modbus_var : ARRAY[0..100] OF INT;
modbus_var_1000 : ARRAY[0..123] OF WORD;
modbus_var_1001 : ARRAY[124..247] OF WORD;
modbus_var_1002 : ARRAY[248..371] OF WORD;
{attribute 'ac_datalog_hysteresis' := '0.2'}
{attribute 'ac_datalog' := 'DatalogChannel_4'}
Temp_chilled_medium_out : REAL;
{attribute 'ac_datalog_hysteresis' := '0.2'}
{attribute 'ac_datalog' := 'DatalogChannel_4'}
Temp_chilled_medium_in : REAL;
{attribute 'ac_datalog_hysteresis' := '0.2'}
{attribute 'ac_datalog' := 'DatalogChannel_4'}
Temp_water_inlet_cond : REAL;
{attribute 'ac_datalog_hysteresis' := '0.2'}
{attribute 'ac_datalog' := 'DatalogChannel_4'}
Press_suction_compr : REAL;
{attribute 'ac_datalog_hysteresis' := '0.5'}
{attribute 'ac_datalog' := 'DatalogChannel_4'}
Press_discharge_compr : REAL;
{attribute 'ac_datalog_hysteresis' := '0.5'}
{attribute 'ac_datalog' := 'DatalogChannel_4'}
Press_oil_receiver : REAL;
{attribute 'ac_datalog_hysteresis' := '0.5'}
{attribute 'ac_datalog' := 'DatalogChannel_4'}
Press_oil_compr : REAL;
{attribute 'ac_datalog_hysteresis' := '0.4'}
{attribute 'ac_datalog' := 'DatalogChannel_4'}
Temp_discharge : REAL;
{attribute 'ac_datalog_hysteresis' := '0.5'}
{attribute 'ac_datalog' := 'DatalogChannel_4'}
Oil_temp_receiver : REAL;
{attribute 'ac_datalog_hysteresis' := '0.5'}
{attribute 'ac_datalog' := 'DatalogChannel_4'}
Max_motor_temp : REAL;
{attribute 'ac_datalog_hysteresis' := '0.2'}
{attribute 'ac_datalog' := 'DatalogChannel_4'}
Temp_motor_bearing_DE : REAL;
{attribute 'ac_datalog_hysteresis' := '0.2'}
{attribute 'ac_datalog' := 'DatalogChannel_4'}
Temp_motor_bearing_NDE : REAL;
{attribute 'ac_datalog_hysteresis' := '4'}
{attribute 'ac_datalog' := 'DatalogChannel_4'}
Motor_current : REAL;
{attribute 'ac_datalog_hysteresis' := '50'}
{attribute 'ac_datalog' := 'DatalogChannel_4'}
Running_hours_comp_unscaled : WORD;
{attribute 'ac_datalog_hysteresis' := '50'}
{attribute 'ac_datalog' := 'DatalogChannel_4'}
Running_hours_oil_pump_unscaled : WORD;
{attribute 'ac_datalog' := 'DatalogChannel_4'}
Anti_recycle_time : REAL;
{attribute 'ac_datalog_hysteresis' := '2'}
{attribute 'ac_datalog' := 'DatalogChannel_4'}
Feedback_compressor : REAL;
{attribute 'ac_datalog_hysteresis' := '0.2'}
{attribute 'ac_datalog' := 'DatalogChannel_4'}
Oil_diff_pressure : REAL;
{attribute 'ac_datalog_hysteresis' := '0.3'}
{attribute 'ac_datalog' := 'DatalogChannel_4'}
Suction_saturated_temp : REAL;
{attribute 'ac_datalog_hysteresis' := '0.2'}
{attribute 'ac_datalog' := 'DatalogChannel_4'}
Discharge_saturated_temp : REAL;
{attribute 'ac_datalog_hysteresis' := '0.2'}
{attribute 'ac_datalog' := 'DatalogChannel_4'}
Temp_water_outlet_cond : REAL;
{attribute 'ac_datalog_hysteresis' := '0.2'}
{attribute 'ac_datalog' := 'DatalogChannel_4'}
Temp_motor_wind_R : REAL;
{attribute 'ac_datalog_hysteresis' := '0.2'}
{attribute 'ac_datalog' := 'DatalogChannel_4'}
Temp_motor_wind_S : REAL;
{attribute 'ac_datalog_hysteresis' := '0.2'}
{attribute 'ac_datalog' := 'DatalogChannel_4'}
Temp_motor_wind_T : REAL;
{attribute 'ac_datalog_hysteresis' := '0.2'}
{attribute 'ac_datalog' := 'DatalogChannel_4'}
Temp_motor_air : REAL;
{attribute 'ac_datalog_hysteresis' := '0.04'}
{attribute 'ac_datalog' := 'DatalogChannel_4'}
dP_CW : REAL;
{attribute 'ac_datalog_hysteresis' := '0.04'}
{attribute 'ac_datalog' := 'DatalogChannel_4'}
dP_SW : REAL;
{attribute 'ac_datalog_hysteresis' := '4'}
{attribute 'ac_datalog' := 'DatalogChannel_4'}
Chiller_capacity : REAL;
{attribute 'ac_datalog_hysteresis' := '2'}
{attribute 'ac_datalog' := 'DatalogChannel_4'}
Temp_oil_inlet_compr : REAL;
Spare : REAL;
{attribute 'ac_datalog_hysteresis' := '2'}
{attribute 'ac_datalog' := 'DatalogChannel_4'}
SP_CW_controller : REAL;
{attribute 'ac_datalog_hysteresis' := '2'}
{attribute 'ac_datalog' := 'DatalogChannel_4'}
Setpoint_oil_pump : REAL;
{attribute 'ac_datalog_hysteresis' := '0.02'}
{attribute 'ac_datalog' := 'DatalogChannel_4'}
Thrust_bearing_position : REAL;
{attribute 'ac_datalog_hysteresis' := '50'}
{attribute 'ac_datalog' := 'DatalogChannel_4'}
Oil_pump_running_hours : REAL;
{attribute 'ac_datalog_hysteresis' := '5'}
{attribute 'ac_datalog' := 'DatalogChannel_4'}
Liquid_level_condenser : REAL;
{attribute 'ac_datalog_hysteresis' := '0.05'}
{attribute 'ac_datalog' := 'DatalogChannel_4'}
Oil_Filter_Drop : REAL; 
{attribute 'ac_datalog_hysteresis' := '2'}
{attribute 'ac_datalog' := 'DatalogChannel_4'}
Proximitor_thrust_pos : REAL;
{attribute 'ac_datalog_hysteresis' := '0.4'}
{attribute 'ac_datalog' := 'DatalogChannel_4'}
Press_chilled_medium_in : REAL;
{attribute 'ac_datalog_hysteresis' := '0.2'}
{attribute 'ac_datalog' := 'DatalogChannel_4'}
Press_water_cond_out : REAL;
{attribute 'ac_datalog_hysteresis' := '0.02'}
{attribute 'ac_datalog' := 'DatalogChannel_4'}
Feedback_sea_water_valve : REAL;
{attribute 'ac_datalog_hysteresis' := '1'}
{attribute 'ac_datalog' := 'DatalogChannel_4'}
Oil_pressure_before_filter : REAL;
{attribute 'ac_datalog_hysteresis' := '0.2'}
{attribute 'ac_datalog' := 'DatalogChannel_4'}
Trafo_winding_temp : REAL;
{attribute 'ac_datalog_hysteresis' := '1'}
{attribute 'ac_datalog' := 'DatalogChannel_4'}
Feedback_VGD : REAL;
{attribute 'ac_datalog_hysteresis' := '4'}
{attribute 'ac_datalog' := 'DatalogChannel_4'}
Feedback_liquid_valve : REAL;
{attribute 'ac_datalog_hysteresis' := '3'}
{attribute 'ac_datalog' := 'DatalogChannel_4'}
Feedback_HGV : REAL;
{attribute 'ac_datalog_hysteresis' := '2'}
{attribute 'ac_datalog' := 'DatalogChannel_4'}
Discharge_superheat : REAL;
{attribute 'ac_datalog_hysteresis' := '0.6'}
{attribute 'ac_datalog' := 'DatalogChannel_4'}
Frequency_oil_pump : REAL;
{attribute 'ac_datalog_hysteresis' := '3'}
{attribute 'ac_datalog' := 'DatalogChannel_4'}
Hot_gas_valve_output : REAL;
{attribute 'ac_datalog_hysteresis' := '2'}
{attribute 'ac_datalog' := 'DatalogChannel_4'}
Control_signal_unit_d : REAL;
{attribute 'ac_datalog_hysteresis' := '2'}
{attribute 'ac_datalog' := 'DatalogChannel_4'}
Stall_detector : REAL;
{attribute 'ac_datalog_hysteresis' := '0.2'}
{attribute 'ac_datalog' := 'DatalogChannel_4'}
SP_MC_controller : REAL;
{attribute 'ac_datalog_hysteresis' := '2'}
{attribute 'ac_datalog' := 'DatalogChannel_4'}
Prerotary_output : REAL;
{attribute 'ac_datalog_hysteresis' := '2'}
{attribute 'ac_datalog' := 'DatalogChannel_4'}
VGD_output : REAL;
{attribute 'ac_datalog_hysteresis' := '2'}
{attribute 'ac_datalog' := 'DatalogChannel_4'}
SP_PID_compressor : REAL;
{attribute 'ac_datalog_hysteresis' := '2'}
{attribute 'ac_datalog' := 'DatalogChannel_4'}
Output_PID_suction : REAL;
{attribute 'ac_datalog_hysteresis' := '2'}
{attribute 'ac_datalog' := 'DatalogChannel_4'}
Output_PID_discharge : REAL;
{attribute 'ac_datalog_hysteresis' := '2'}
{attribute 'ac_datalog' := 'DatalogChannel_4'}
Output_PID_motor : REAL;
{attribute 'ac_datalog_hysteresis' := '2'}
{attribute 'ac_datalog' := 'DatalogChannel_4'}
Output_PID_superheat : REAL;
{attribute 'ac_datalog_hysteresis' := '2'}
{attribute 'ac_datalog' := 'DatalogChannel_4'}
SP_control : REAL;
{attribute 'ac_datalog_hysteresis' := '2'}
{attribute 'ac_datalog' := 'DatalogChannel_4'}
Unit_control_signal : REAL;
{attribute 'ac_datalog_hysteresis' := '2'}
{attribute 'ac_datalog' := 'DatalogChannel_4'}
Feedback_PRV : REAL;
{attribute 'ac_datalog_hysteresis' := '0.3'}
{attribute 'ac_datalog' := 'DatalogChannel_4'}
Theta_out : REAL;
{attribute 'ac_datalog_hysteresis' := '50'}
{attribute 'ac_datalog' := 'DatalogChannel_4'}
Alarm_limit_stall_count_unscaled : WORD;
{attribute 'ac_datalog_hysteresis' := '50'}
{attribute 'ac_datalog' := 'DatalogChannel_4'}
Alarm_limit_stall_count : REAL;
{attribute 'ac_datalog_hysteresis' := '2'}
{attribute 'ac_datalog' := 'DatalogChannel_4'}
Stall_ramp : REAL;
Min_allowed_PRVposition : REAL;
Number_of_starts : REAL;
SP_freq_oil_pump_VFD : REAL;
SP_oil_pressure_diff : REAL;
SP_oil_pressure : REAL;
{attribute 'ac_datalog_hysteresis' := '2'}
{attribute 'ac_datalog' := 'DatalogChannel_4'}
Setpoint_conv_oil_pump : REAL;
Days_above_stall_limit : REAL;
Hrs_above_stall_limit : REAL;
Min_above_stall_limit : REAL;
Sec_above_stall_limit : REAL;
{attribute 'ac_datalog_hysteresis' := '2'}
{attribute 'ac_datalog' := 'DatalogChannel_4'}
SP_cond_press : REAL;
{attribute 'ac_datalog_hysteresis' := '2'}
{attribute 'ac_datalog' := 'DatalogChannel_4'}
SP_PID_Level : REAL;
{attribute 'ac_datalog_hysteresis' := '2'}
{attribute 'ac_datalog' := 'DatalogChannel_4'}
Control_signal_SW_valve : REAL;
{attribute 'ac_datalog_hysteresis' := '4'}
{attribute 'ac_datalog' := 'DatalogChannel_4'}
Liquid_valve_output : REAL;
{attribute 'ac_datalog_hysteresis' := '0.2'}
{attribute 'ac_datalog' := 'DatalogChannel_4'}
SP_PID_seawater : REAL;
{attribute 'ac_datalog_hysteresis' := '4'}
{attribute 'ac_datalog' := 'DatalogChannel_4'}
Chiller_capacity_t1 : REAL;
{attribute 'ac_datalog_hysteresis' := '2'}
{attribute 'ac_datalog' := 'DatalogChannel_4'}
SW_pump_speed_order : REAL;
{attribute 'ac_datalog_hysteresis' := '0.4'}
{attribute 'ac_datalog' := 'DatalogChannel_4'}
Press_chilled_medium_out : REAL;
{attribute 'ac_datalog_hysteresis' := '50'}
{attribute 'ac_datalog' := 'DatalogChannel_4'}
Running_hours_compressormotor : REAL;
{attribute 'ac_datalog_hysteresis' := '0.2'}
{attribute 'ac_datalog' := 'DatalogChannel_4'}
Press_water_cond_inlet : REAL;
{attribute 'ac_datalog_hysteresis' := '2'}
{attribute 'ac_datalog' := 'DatalogChannel_4'}
Speed_feedback_VFD : REAL;
{attribute 'ac_datalog_hysteresis' := '2'}
{attribute 'ac_datalog' := 'DatalogChannel_4'}
Order_VFD_perc : REAL;
{attribute 'ac_datalog_hysteresis' := '2'}
{attribute 'ac_datalog' := 'DatalogChannel_4'}
Order_VFD_Hz : REAL;
{attribute 'ac_datalog_hysteresis' := '2'}
{attribute 'ac_datalog' := 'DatalogChannel_4'}
Temp_trafo_wind_U : REAL;
{attribute 'ac_datalog_hysteresis' := '0.2'}
{attribute 'ac_datalog' := 'DatalogChannel_4'}
Temp_trafo_wind_V : REAL;
{attribute 'ac_datalog_hysteresis' := '0.2'}
{attribute 'ac_datalog' := 'DatalogChannel_4'}
Temp_trafo_wind_W : REAL;
{attribute 'ac_datalog_hysteresis' := '2'}
{attribute 'ac_datalog' := 'DatalogChannel_4'}
Opt_speed_VFD_perc : REAL;
{attribute 'ac_datalog_hysteresis' := '2'}
{attribute 'ac_datalog' := 'DatalogChannel_4'}
Opt_speed_VFD_Hz : REAL;
Surge_counter_VFD : REAL;
Spare_4 : REAL;
Spare_3 : REAL;
Spare_2 : REAL;
Spare_0 : REAL;
Vibration_compressor_DE: REAL;
Vibration_compressor_NDE: REAL;
Feedback_seawater_valve_overboard : REAL;
Feedback_seawater_valve_bypass : REAL;
CW_flow_m3: REAL;
SW_flow_m3: REAL;
Max_motor_wind_temp: REAL;
Order_SWW_overboard: REAL;
Order_SWW_bypass: REAL;
{attribute 'ac_datalog_hysteresis' := '0.4'}
{attribute 'ac_datalog' := 'DatalogChannel'}
COP_chiller_mech : REAL ;
{attribute 'ac_datalog_hysteresis' := '50'}
{attribute 'ac_datalog' := 'DatalogChannel'}
P2_mot_1_kW : REAL ;
{attribute 'ac_datalog_hysteresis' := '50'}
{attribute 'ac_datalog' := 'DatalogChannel'}
P1_motor_kW : REAL ;
{attribute 'ac_datalog_hysteresis' := '0.4'}
{attribute 'ac_datalog' := 'DatalogChannel'}
COP_chiller_ele : REAL ;
{attribute 'ac_datalog_hysteresis' := '0.2'}
{attribute 'ac_datalog' := 'DatalogChannel'}
PI_chiller : REAL ;
;{attribute 'ac_datalog_hysteresis' := '40'}
{attribute 'ac_datalog' := 'DatalogChannel'}
Wasted_energy_kW : REAL ;
{attribute 'ac_datalog_hysteresis' := '200'}
{attribute 'ac_datalog' := 'DatalogChannel'}
Chiller_capacity_kW : REAL;
Thrust_bearing_ref_min : REAL ;
Thrust_bearing_ref_max : REAL ;
Thrust_bearing_ref : REAL ;
Q2_chillerMWh : REAL ;
Chiller_P1_MWh : REAL ;
Cal_date_MMYY : REAL ;
Chiller_P2_MWh : REAL ;
Liquid_line_temp : REAL ;
VFD_motor_current : REAL ;
Feedback_liquid_valve_raw : REAL ;
Feedback_VGD_raw : REAL ;
Feedback_PRV_raw : REAL ;
Feedback_HGV_raw : REAL ;
Feedback_seawater_valve_overboard_raw : REAL ;
Feedback_seawater_valve_bypass_raw : REAL ;
SP_cond_press_limit : REAL ;
SP_evap_press_limit : REAL ;
SP_discharge_superheat_limit : REAL ;
SP_t1 : REAL ;
VFD_min_allowed_frequence : REAL ;
VFD_min_allowed_speed : REAL ;

Trip_BITs_0_to_15 : WORD;
Trip_BITs_16_to_31: WORD;
Trip_BITs_32_to_47: WORD;
Trip_BITs_48_to_63: WORD;
Trip_BITs_64_to_79: WORD;
Trip_BITs_80_to_95: WORD;
Trip_BITs_96_to_121: WORD;
Trip_BITs_122_to_137: WORD;
Trip_BITs_138_to_153: WORD;
Trip_BITs_154_to_169: WORD;
Trip_BITs_170_to_185: WORD;
Trip_BITs_186_to_201: WORD;


Alarm_BITs_0_to_15: WORD;
Alarm_BITs_16_to_31: WORD;
Alarm_BITs_32_to_47: WORD;
Alarm_BITs_48_to_63: WORD;
Alarm_BITs_64_to_79: WORD;
Alarm_BITs_80_to_95: WORD;
Alarm_BITs_96_to_111: WORD;

Status_BITs_0_to_15 : WORD;
Status_BITs_16_to_31 : WORD;
Status_BITs_32_to_47: WORD;
Status_BITs_48_to_63: WORD;
Status_BITs_64_to_79: WORD;
Status_BITs_80_to_95: WORD;
Status_BITs_96_to_111: WORD;
Status_BITs_112_to_127: WORD;




DI_Status_BITs_0_to_15 : WORD;
DI_Status_BITs_16_to_31: WORD;

DO_Status_BITs_16_to_31: WORD;
DO_Status_BITs_32_to_47: WORD;

T_Overload_compressor_motor : BOOL;
T_Compressor_running_failure : BOOL;
T_Low_chilled_medium_outlet : BOOL;
T_Low_sea_water_flow : BOOL;
T_Oil_level_motor_bearing : BOOL;

T_Low_oil_flow : BOOL;
T_Overload_oil_pump_motor : BOOL;
T_Oil_pump_running_failure : BOOL;
T_Low_oil_flow_trip : BOOL;
T_High_temp_oil_receiver : BOOL;
T_Low_temp_oil_receiver : BOOL;
T_Low_suction_pressure : BOOL;
T_High_suction_pressure : BOOL;
T_High_discharge_pressure : BOOL;
T_Low_discharge_pressure : BOOL;
T_High_discharge_temp : BOOL;
T_Low_oil_diff_pressure : BOOL;
T_High_diff_oil_pressure : BOOL;
T_Starting_to_long : BOOL;
T_Surge_detection : BOOL;
T_Comp_thrust_bearing_position : BOOL;
Spare_trip_1 : BOOL;
T_Chilled_pump_run_failure : BOOL;
T_Sea_water_pump_run_failure : BOOL;
T_Low_chilled_medium_flow : BOOL;
T_High_chilled_medium_flow : BOOL;
T_Low_condenser_flow : BOOL;
T_High_condenser_flow : BOOL;
T_Emergency_stop : BOOL;
T_High_comp_mot_DE_bear_temp : BOOL;
T_High_comp_mot_NDE_bear_temp : BOOL;
T_High_motor_air_temp : BOOL;
T_Comp_motor_leak_detection : BOOL;
T_High_comp_mot_DE_bear_vib : BOOL;
T_High_comp_mot_NDE_bear_Vib : BOOL;
T_High_comp_motor_wind_temp : BOOL;
Spare_trip_2 : BOOL;
T_Rotating_stall_trip : BOOL;
T_Analog_inputs : BOOL;
T_Feedback_CW_valve : BOOL;
T_Low_oil_diff_press_prelub : BOOL;
T_Low_oil_diff_press_standstil : BOOL;

T_Spare_3 : BOOL;
T_Spare_4 : BOOL;
T_Spare_5 : BOOL;
T_Spare_6 : BOOL;
T_Spare_7 : BOOL;
T_Spare_8 : BOOL;
T_High_temp_oil_inlet_comp : BOOL;
T_Comp_motor_power_loss : BOOL;
Spare_trip_3 : BOOL;
T_Cathodic_protect_sys_alarm : BOOL;
T_High_oil_filter_diff_press : BOOL;
T_Flow_switch_FT01 : BOOL;
T_Starter_failure_trip : BOOL;
T_Incorrect_feedback_starter_trip : BOOL;

A_VGD_fault : BOOL;
A_High_condenser_flow : BOOL;
A_Rotating_stall : BOOL;
A_High_temp_oil_inlet_comp : BOOL;
SpareAlarm_1 : BOOL;
A_High_motor_air_temp : BOOL;
A_High_control_panel_temp : BOOL;
A_Low_oil_diff_pressure : BOOL;
Spare_alarm_2 : BOOL;
A_High_comp_motor_winding_temp : BOOL;
A_High_comp_mo_DE_bear_temp : BOOL;
A_High_comp_mo_NDE_bear_temp : BOOL;
A_High_comp_mo_DE_bear_vib : BOOL;
A_High_comp_mo_NDE_bear_vib : BOOL;
A_Low_chilled_medium_flow : BOOL;
A_High_chilled_medium_flow : BOOL;
A_Low_sea_water_flow : BOOL;
A_Seawater_pump_not_running : BOOL;
A_Spare : BOOL;
A_Spare_1 : BOOL;
A_Spare_2 : BOOL;
A_Spare_3 : BOOL;
A_Spare_4 : BOOL;
A_Spare_5 : BOOL;
A_Spare_6 : BOOL;
A_Spare_7 : BOOL;
A_Spare_8 : BOOL;
A_Spare_9 : BOOL;
A_Spare_10 : BOOL;
A_Spare_11 : BOOL;
A_High_oil_filter_diff_press : BOOL;
A_Spare_12 : BOOL;
A_Spare_13 : BOOL;
A_Spare_14 : BOOL;
A_Spare_15 : BOOL;
A_Spare_16 : BOOL;
A_Spare_17 : BOOL;
Anti_recycle_status : BOOL;
Low_oil_temperature : BOOL;
Low_oil_temp_auto : BOOL;
Oil_heater : BOOL;
Sea_water_pump : BOOL;
Comp_oil_pump : BOOL;
Bearing_oil_pump : BOOL;
Solenoid_oil_return : BOOL;
Unit_running : BOOL;
Unit_remote : BOOL;
Unit_auto : BOOL;
Unit_manual : BOOL;
Unit_trip : BOOL;
Unit_alarm : BOOL;
Unit_start_switch : BOOL;
Unit_available : BOOL;
Unit_fault : BOOL;
S_Spare_1 : BOOL;
S_Spare_2 : BOOL;
S_Spare_3 : BOOL;
S_Spare_4 : BOOL;
S_Spare_5 : BOOL;
S_Spare_6 : BOOL;
S_Spare_7 : BOOL;
S_Spare_8 : BOOL;
Solenoid_liquid_inj: BOOL;
CW_Flow_ind : BOOL;
Open_chilled_water_valve : BOOL;
Feedback_chilled_water_valve : BOOL;
Open_order_swv_overboard : BOOL;
Close_order_swv_overboard : BOOL;
Open_order_swv_bypass : BOOL;
Close_order_swv_bypass : BOOL;
VFD_man_auto : BOOL ;
VFD_freq_jump_on : BOOL ;
VFD_ramp_100_perc : BOOL ;
VFD_locked_100_perc : BOOL;
VFD_ramp_d_PRVcontrol : BOOL;
PRV_control : BOOL;
VFD_control : BOOL;
VFD_fixed_speed : BOOL;
Spare_151: BOOL;
T_Transformer_winding_temp : BOOL;
A_Transformer_winding_temp : BOOL;
T_trafo_opening_main_breaker : BOOL;
T_VFD : BOOL;
VFD_ready : BOOL;
T_VFD_emergency_stop : BOOL;
T_Low_5VDC_supply : BOOL;
T_High_5VDC_supply : BOOL;
T_Spare_9 : BOOL;
T_Spare_10 : BOOL;
T_Spare_11 : BOOL;
T_Spare_12 : BOOL;
T_Spare_13 : BOOL;
T_Low_liquid_level : BOOL;
T_SW_pump_off_to_long : BOOL;
T_Softstarter_failure : BOOL;
T_Motorstarter_failure : BOOL ;
T_CW_valveopen_failure : BOOL ;
T_SW_valveopen_failure : BOOL ;
T_High_disch_superheat :BOOL ;
T_Low_disch_superheat :BOOL ;
T_High_CW_outlet_temp : BOOL;
T_Low_CW_outlet_temp : BOOL;
T_Low_CW_inlet_temp : BOOL;
T_High_CW_inlet_temp : BOOL;
T_High_SW_outlet_temp : BOOL;
T_Low_SW_outlet_temp : BOOL;
T_Low_SW_inlet_temp : BOOL;
T_High_SW_inlet_temp : BOOL;
T_High_motor_wind_temp_R : BOOL;
T_High_motor_wind_temp_S : BOOL;
T_High_motor_wind_temp_T : BOOL;
T_High_press_ratio : BOOL;
T_Low_press_ratio : BOOL;
T_Low_CW_dP : BOOL;
T_High_CW_dP : BOOL;
T_Low_SW_dP : BOOL;
T_High_SW_dP : BOOL;
T_Long_time_PRV : BOOL;
T_Comp_thrust_neg_move : BOOL;
T_Comp_thrust_pos_move : BOOL;
T_VGD_fault : BOOL;
T_Low_oilpress_prelube : BOOL;
T_Low_temp_oil_inlet_comp : BOOL;
T_Low_oilpress_standby : BOOL;
T_Rotating_stall : BOOL;

T_Sensor_failure_AI_128: BOOL;
T_Sensor_failure_AI_130: BOOL;
T_Sensor_failure_AI_134: BOOL;
T_Sensor_failure_AI_256: BOOL;
T_Sensor_failure_AI_258: BOOL;
T_Sensor_failure_AI_260: BOOL;
T_Sensor_failure_AI_262: BOOL;
T_Sensor_failure_AI_264: BOOL;
T_Sensor_failure_AI_266: BOOL;
T_Sensor_failure_AI_268: BOOL;
T_Sensor_failure_AI_270: BOOL;
T_Sensor_failure_AI_272: BOOL;
T_Sensor_failure_AI_274: BOOL;
T_Sensor_failure_AI_276: BOOL;
T_Sensor_failure_AI_278: BOOL;
T_Sensor_failure_AI_280: BOOL;
T_Sensor_failure_AI_282: BOOL;
T_Sensor_failure_AI_284: BOOL;
T_Sensor_failure_AI_286: BOOL;
T_Sensor_failure_AI_288: BOOL;
T_Sensor_failure_AI_290: BOOL;
T_Sensor_failure_AI_292: BOOL;
T_Sensor_failure_AI_294: BOOL;
T_Sensor_failure_AI_296: BOOL;
T_Sensor_failure_AI_298: BOOL;
T_Sensor_failure_AI_330: BOOL;
T_Sensor_failure_AI_320: BOOL;
T_Sensor_failure_AI_322: BOOL;
T_Sensor_failure_AI_324: BOOL;
T_Sensor_failure_AI_326: BOOL;
T_Sensor_failure_AI_328: BOOL;
T_Sensor_failure_AI_332: BOOL;
T_Sensor_failure_AI_334: BOOL;
T_Sensor_failure_AI_300: BOOL;
T_Sensor_failure_AI_302: BOOL;
T_Sensor_failure_AI_304: BOOL;
T_Sensor_failure_AI_306: BOOL;
T_Sensor_failure_AI_308: BOOL;
T_Sensor_failure_AI_310: BOOL;
T_Sensor_failure_AI_312: BOOL;
T_Sensor_failure_AI_314: BOOL;
T_Sensor_failure_AI_316: BOOL;
T_Sensor_failure_AI_318: BOOL;
T_Sensor_failure_AI_352: BOOL;
T_Sensor_failure_AI_354: BOOL;
T_Sensor_failure_AI_360: BOOL;
T_Sensor_failure_AI_362: BOOL;
T_Sensor_failure_AI_364: BOOL;
T_Sensor_failure_AI_368: BOOL;
T_Sensor_failure_AI_370: BOOL;
T_Sensor_failure_AI_372: BOOL;
T_Sensor_failure_AI_374: BOOL;
T_Sensor_failure_AI_376: BOOL;
T_Sensor_failure_AI_378: BOOL;
T_Sensor_failure_AI_380: BOOL;
T_Sensor_failure_AI_382: BOOL;
T_Sensor_failure_AI_336: BOOL;
T_Sensor_failure_AI_338: BOOL;
T_Sensor_failure_AI_340: BOOL;
T_Sensor_failure_AI_342: BOOL;
T_Sensor_failure_AI_344: BOOL;
T_Sensor_failure_AI_346: BOOL;
T_Sensor_failure_AI_348: BOOL;
T_Sensor_failure_AI_350: BOOL;
T_Sensor_failure_AI_752: BOOL;
T_Sensor_failure_AI_754: BOOL;
T_Sensor_failure_AI_756: BOOL;
T_Sensor_failure_AI_760: BOOL;
T_Sensor_failure_AI_772: BOOL;
T_Sensor_failure_AI_774: BOOL;
T_Sensor_failure_AI_776: BOOL;
T_Sensor_failure_AI_778: BOOL;
T_Sensor_failure_AI_780: BOOL;

A_high_disch_press : BOOL ;
A_low_disch_press : BOOL ;
A_Low_suction_pressure : BOOL;
A_High_suction_pressure : BOOL;
A_High_discharge_temp : BOOL;
A_High_oil_temp_receiver : BOOL;
A_Low_oil_temp_receiver : BOOL;
A_Low_temp_oil_inlet_comp : BOOL;
A_High_oil_diff_pressure : BOOL;
A_Low_discharge_superheat : BOOL;
A_High_discharge_superheat : BOOL;
A_Low_CW_outlet_temp : BOOL;
A_High_CW_outlet_temp : BOOL;
A_Low_CW_inlet_temp : BOOL;
A_High_CW_inlet_temp : BOOL;
A_High_SW_outlet_temp : BOOL;
A_Low_condenser_flow : BOOL;
A_High_press_ratio : BOOL;
A_Low_press_ratio : BOOL;
A_Motor_speed_low : BOOL;
A_Low_SW_outlet_temp : BOOL;
A_Low_SW_inlet_temp : BOOL;
A_High_SW_inlet_temp : BOOL;
A_High_suction_superheat : BOOL;
A_Low_suction_superheat : BOOL;
A_High_temp_oil_separator : BOOL;
A_Low_temp_oil_separator : BOOL;
A_High_motor_wind_temp_R : BOOL;
A_High_motor_wind_temp_S : BOOL;
A_High_motor_wind_temp_T : BOOL;
A_High_CW_dP : BOOL;
A_Low_CW_dP : BOOL;
A_High_SW_dP : BOOL;
A_Low_SW_dP : BOOL;

Start_inhib_time_between_Start : BOOL;
Start_inhib_time_beetween_Stop : BOOL;
Start_inhib_PRV_not_min : BOOL;
Start_inhib_Motor_overload : BOOL;
Remote_bilge_pump_control : BOOL;
CW_pump_running : BOOL;
A_Low_liquid_level : BOOL;
A_Suction_press_limit : BOOL;
A_Discharge_press_limit : BOOL;
A_Discharge_superheat_limit : BOOL;
A_Motor_current_limit : BOOL;


DI_0_0_Emergency_stop : BOOL;
DI_0_0 : BOOL;
DI_0_1 : BOOL;
DI_0_2_Fault_reset : BOOL;
DI_0_2 : BOOL;
DI_0_3 : BOOL;
DI_0_4 : BOOL;
DI_0_5 : BOOL;
DI_0_6_Overload_protection : BOOL;
DI_0_6 : BOOL;
DI_0_7 : BOOL;
DI_1_0_Overload_oilpump : BOOL;
DI_1_0 : BOOL;
DI_1_1 : BOOL;
DI_1_2 : BOOL;
DI_1_3 : BOOL;
Power_available : BOOL;
DI_1_4 : BOOL;
DI_1_5_Starter_failure : BOOL;
DI_1_5 : BOOL;
DI_8_0_Controlpanel_temp : BOOL;
DI_8_0 : BOOL;
DI_8_1 : BOOL;
DI_8_2_VGD_limit_switch : BOOL;
DI_8_2 : BOOL;
DI_8_3_water_leak_motor  : BOOL;
DI_8_3 : BOOL;
DI_8_4_Catodic_protection : BOOL;
DI_8_4 : BOOL;
DI_8_5_Trust_bearing_probe : BOOL;
DI_8_5 : BOOL;
DI_8_6_ESD_operation : BOOL;
DI_8_6 : BOOL;
DI_8_7 : BOOL;
DI_9_0_MV_breaker_available : BOOL;
DI_9_0 : BOOL;
DI_9_1 : BOOL;
DI_9_2_Safe_return_to_port : BOOL;
DI_9_2 : BOOL;
DI_9_3 : BOOL;
DI_9_4_VFD_emergency_stop : BOOL;
DI_9_4 : BOOL;
DI_9_5 : BOOL;
DI_9_6 : BOOL;
DI_9_7 : BOOL;
DO_0_0_Start_signal_comp : BOOL;
DO_0_0 : BOOL;
DO_0_1_Start_signal_oil_pump : BOOL;
DO_0_1 : BOOL;
DO_0_2_Start_signal_SW_pump : BOOL;
DO_0_2 : BOOL;
DO_0_3_Start_signal_CW_pump : BOOL;
DO_0_3 : BOOL;
DO_0_4_Solenoid_valve_oil : BOOL;
DO_0_4 : BOOL;
DO_0_5_Solenoid_valve_liquid : BOOL;
DO_0_5 : BOOL;
DO_0_6_Oil_heater : BOOL;
DO_0_6 : BOOL;
DO_0_7_Comp_heater : BOOL;
DO_0_7 : BOOL;
DO_1_0 : BOOL;
DO_1_1 : BOOL;
DO_8_0_Liquid_valve_open : BOOL;
DO_8_0 : BOOL;
DO_8_1_Liquid_valve_close : BOOL;
DO_8_1 : BOOL;
DO_8_2_VGD_open : BOOL;
DO_8_2 : BOOL;
DO_8_3_VGD_close : BOOL;
DO_8_3 : BOOL;
DO_8_4_PRV_open : BOOL;
DO_8_4 : BOOL;
DO_8_5_PRV_close : BOOL;
DO_8_5 : BOOL;
DO_8_6_HGV_open : BOOL;
DO_8_6 : BOOL;
DO_8_7_HGV_close : BOOL;
DO_8_7 : BOOL;
DO_9_0_Open_order_swv_overboard : BOOL;
DO_9_0 : BOOL;
DO_9_1_Close_order_swv_overboard : BOOL;
DO_9_1 : BOOL;
DO_9_2_Open_order_swv_bypass : BOOL;
DO_9_2 : BOOL;
DO_9_3_Close_order_swv_bypass : BOOL;
DO_9_3 : BOOL;
DO_9_4 : BOOL;
DO_9_5 : BOOL;
DO_9_6 : BOOL;
DO_9_7 : BOOL;
Power_request : BOOL;
DO_12_0 : BOOL;
DO_12_1_Compressor_ready : BOOL;
DO_12_1 : BOOL;
DO_12_2 : BOOL;
DO_12_3 : BOOL;
DO_12_4_Control_panel_alarm : BOOL;
DO_12_4 : BOOL;
DO_12_5_Auto_reset : BOOL;
DO_12_5 : BOOL;
DO_12_6_Unit_running : BOOL;
DO_12_6 : BOOL;
DO_12_7 : BOOL;
Start_inhib_time_Oil_receiver_temp : BOOL;
PrV_in_min : BOOL;


//Graphic variables
Unit_switch_status : INT;
i : INT;
show_trendvalue : ARRAY[0..50] OF BOOL;
select_trendvalue : INT :=0 ;

END_VAR


Temp_chilled_medium_out:=scaleFunction(modbus_var_1000[10],0.1, 0);
Temp_chilled_medium_in:=scaleFunction(modbus_var_1000[11],0.1, 0);
Temp_water_inlet_cond:=scaleFunction(modbus_var_1000[12],0.1, 0);
Press_suction_compr:=scaleFunction(modbus_var_1000[13],0.01, 0);
Press_discharge_compr:=scaleFunction(modbus_var_1000[14],0.01, 0);
Press_oil_receiver:=scaleFunction(modbus_var_1000[15],0.01, 0);
Press_oil_compr:=scaleFunction(modbus_var_1000[16],0.01, 0);
Temp_discharge:=scaleFunction(modbus_var_1000[17],0.1, 0);
Oil_temp_receiver:=scaleFunction(modbus_var_1000[18],0.1, 0);
Max_motor_temp:=scaleFunction(modbus_var_1000[19],0.1, 0);
Temp_motor_bearing_DE:=scaleFunction(modbus_var_1000[20],0.1, 0);
Temp_motor_bearing_NDE:=scaleFunction(modbus_var_1000[21],0.1, 0);
Motor_current:=scaleFunction(modbus_var_1000[22],1.0, 0);
Running_hours_comp_unscaled:=modbus_var_1000[23];
//Anti_recycle_time:=scaleFunction(modbus_var_1000[24],1.0, 0);
Feedback_compressor:=scaleFunction(modbus_var_1000[25],1.0, 0);
Oil_diff_pressure:=scaleFunction(modbus_var_1000[26],0.01, 0);
Suction_saturated_temp:=scaleFunction(modbus_var_1000[27],0.1, 0);
Discharge_saturated_temp:=scaleFunction(modbus_var_1000[28],0.1, 0);
Temp_water_outlet_cond:=scaleFunction(modbus_var_1000[29],0.1, 0);
Temp_motor_wind_R:=scaleFunction(modbus_var_1000[30],0.1, 0);
Temp_motor_wind_S:=scaleFunction(modbus_var_1000[31],0.1, 0);
Temp_motor_wind_T:=scaleFunction(modbus_var_1000[32],0.1, 0);
Temp_motor_air:=scaleFunction(modbus_var_1000[33],0.1, 0);
dP_CW:=scaleFunction(modbus_var_1000[34],0.01, 0);
dP_SW:=scaleFunction(modbus_var_1000[35],0.01, 0);
CW_flow_m3:=scaleFunction(modbus_var_1000[36],1.0, 0);
Temp_oil_inlet_compr:=scaleFunction(modbus_var_1000[37],0.1, 0);
Stall_detector:=scaleFunction(modbus_var_1000[38],0.01, 0);
SP_CW_controller:=scaleFunction(modbus_var_1000[39],0.1, 0);
Feedback_sea_water_valve:=scaleFunction(modbus_var_1000[40],0.1, 0);
Oil_pressure_before_filter:=scaleFunction(modbus_var_1000[41],0.01, 0);
Feedback_VGD:=scaleFunction(modbus_var_1000[42],0.1, 0);
Chiller_capacity:=scaleFunction(modbus_var_1000[43],0.1, 0);
Setpoint_oil_pump:=scaleFunction(modbus_var_1000[44],0.01, 0);
Thrust_bearing_position:=scaleFunction(modbus_var_1000[45],0.1, 0);
Oil_pump_running_hours:=scaleFunction(modbus_var_1000[46],10, 0);
Liquid_level_condenser:=scaleFunction(modbus_var_1000[47],0.1, 0);
Oil_Filter_Drop:=scaleFunction(modbus_var_1000[48],0.01, 0);
Proximitor_thrust_pos:=scaleFunction(modbus_var_1000[49],0.1, 0);
//Spare_old_write_bits:=scaleFunction(modbus_var_1000[50],1.0, 0);
Press_chilled_medium_in:=scaleFunction(modbus_var_1000[51],0.01, 0);
Press_water_cond_out:=scaleFunction(modbus_var_1000[52],0.01, 0);
Discharge_superheat:=scaleFunction(modbus_var_1000[53],0.1, 0);
Frequency_oil_pump:=scaleFunction(modbus_var_1000[54],0.1, 0);
Feedback_liquid_valve:=scaleFunction(modbus_var_1000[55],0.1, 0);
Hot_gas_valve_output:=scaleFunction(modbus_var_1000[56],0.1, 0);
Control_signal_unit_d:=scaleFunction(modbus_var_1000[57],0.1, 0);
SP_MC_controller:=scaleFunction(modbus_var_1000[58],0.1, 0);
Prerotary_output:=scaleFunction(modbus_var_1000[59],0.1, 0);
VGD_output:=scaleFunction(modbus_var_1000[60],0.1, 0);
SP_PID_compressor:=scaleFunction(modbus_var_1000[61],0.1, 0);
Output_PID_suction:=scaleFunction(modbus_var_1000[62],0.1, 0);
Output_PID_discharge:=scaleFunction(modbus_var_1000[63],0.1, 0);
Output_PID_motor:=scaleFunction(modbus_var_1000[64],0.1, 0);
Output_PID_superheat:=scaleFunction(modbus_var_1000[65],0.1, 0);
SP_control:=scaleFunction(modbus_var_1000[66],0.1, 0);
Unit_control_signal:=scaleFunction(modbus_var_1000[67],0.1, 0);
Feedback_PRV:=scaleFunction(modbus_var_1000[68],0.1, 0);
Theta_out:=scaleFunction(modbus_var_1000[69],0.1, 0);
Alarm_limit_stall_count:=scaleFunction(modbus_var_1000[70],1.0, 0);
Stall_ramp:=scaleFunction(modbus_var_1000[71],0.1, 0);
Min_allowed_PRVposition:=scaleFunction(modbus_var_1000[72],0.1, 0);
Number_of_starts:=scaleFunction(modbus_var_1000[73],1.0, 0);
SP_oil_pressure:=scaleFunction(modbus_var_1000[74],0.01, 0);
Setpoint_conv_oil_pump:=scaleFunction(modbus_var_1000[75],0.1, 0);
Days_above_stall_limit:=scaleFunction(modbus_var_1000[76],1.0, 0);
Hrs_above_stall_limit:=scaleFunction(modbus_var_1000[77],1.0, 0);
Min_above_stall_limit:=scaleFunction(modbus_var_1000[78],1.0, 0);
Sec_above_stall_limit:=scaleFunction(modbus_var_1000[79],1.0, 0);
SP_PID_Level:=scaleFunction(modbus_var_1000[80],0.1, 0);
Control_signal_SW_valve:=scaleFunction(modbus_var_1000[81],0.1, 0);
Feedback_HGV:=scaleFunction(modbus_var_1000[82],0.1, 0);
Liquid_valve_output:=scaleFunction(modbus_var_1000[83],0.1, 0);
SP_PID_seawater:=scaleFunction(modbus_var_1000[84],0.1, 0);
Chiller_capacity_t1:=scaleFunction(modbus_var_1000[85],0.1, 0);
SW_pump_speed_order:=scaleFunction(modbus_var_1000[86],0.1, 0);
Anti_recycle_time:=scaleFunction(modbus_var_1000[87],1.0, 0);
Press_chilled_medium_out:=scaleFunction(modbus_var_1000[88],0.01, 0);
Press_water_cond_inlet:=scaleFunction(modbus_var_1000[89],0.01, 0);
Running_hours_compressormotor:=scaleFunction(modbus_var_1000[90],10, 0);

Trip_BITs_0_to_15:=modbus_var_1000[0];
Trip_BITs_16_to_31:=modbus_var_1000[1];
Trip_BITs_32_to_47:=modbus_var_1000[2];
Trip_BITs_48_to_63:=modbus_var_1000[3];
Trip_BITs_64_to_79:=modbus_var_1000[4];
// Alarm_BITs_80_to_95:=modbus_var_1000[5];
// Alarm_BITs_96_to_111:=modbus_var_1000[6];
Status_BITs_0_to_15:=modbus_var_1000[5];
Status_BITs_16_to_31:=modbus_var_1000[6];

T_Low_suction_pressure:=maskbitFunction(Trip_BITs_0_to_15,0);
T_High_discharge_pressure:=maskbitFunction(Trip_BITs_0_to_15,1);
T_High_discharge_temp:=maskbitFunction(Trip_BITs_0_to_15,2);
T_Low_oil_diff_pressure:=maskbitFunction(Trip_BITs_0_to_15,3);
T_High_diff_oil_pressure:=maskbitFunction(Trip_BITs_0_to_15,4);
T_Starting_to_long:=maskbitFunction(Trip_BITs_0_to_15,5);
T_Surge_detection:=maskbitFunction(Trip_BITs_0_to_15,6);
T_Comp_thrust_bearing_position:=maskbitFunction(Trip_BITs_0_to_15,7);
T_Overload_compressor_motor:=maskbitFunction(Trip_BITs_0_to_15,8);
T_Compressor_running_failure:=maskbitFunction(Trip_BITs_0_to_15,9);
T_Low_chilled_medium_outlet:=maskbitFunction(Trip_BITs_0_to_15,10);
T_Low_oil_flow:=maskbitFunction(Trip_BITs_0_to_15,11);
T_Overload_oil_pump_motor:=maskbitFunction(Trip_BITs_0_to_15,12);
T_Oil_pump_running_failure:=maskbitFunction(Trip_BITs_0_to_15,13);
T_Low_oil_flow_trip:=maskbitFunction(Trip_BITs_0_to_15,14);
T_High_temp_oil_receiver:=maskbitFunction(Trip_BITs_0_to_15,15);
T_High_comp_motor_wind_temp:=maskbitFunction(Trip_BITs_16_to_31,0);
T_High_comp_mot_DE_bear_temp:=maskbitFunction(Trip_BITs_16_to_31,1);
T_High_comp_mot_NDE_bear_temp:=maskbitFunction(Trip_BITs_16_to_31,2);
T_High_motor_air_temp:=maskbitFunction(Trip_BITs_16_to_31,3);
T_Comp_motor_leak_detection:=maskbitFunction(Trip_BITs_16_to_31,4);
T_High_5VDC_supply:=maskbitFunction(Trip_BITs_16_to_31,5);
T_Low_5VDC_supply:=maskbitFunction(Trip_BITs_16_to_31,6);
T_Chilled_pump_run_failure:=maskbitFunction(Trip_BITs_16_to_31,7);
T_Sea_water_pump_run_failure:=maskbitFunction(Trip_BITs_16_to_31,8);
T_Low_chilled_medium_flow:=maskbitFunction(Trip_BITs_16_to_31,9);
T_High_chilled_medium_flow:=maskbitFunction(Trip_BITs_16_to_31,10);
T_Low_sea_water_flow:=maskbitFunction(Trip_BITs_16_to_31,11);
T_High_condenser_flow:=maskbitFunction(Trip_BITs_16_to_31,12);
A_High_temp_oil_inlet_comp:=maskbitFunction(Trip_BITs_16_to_31,13);
T_Comp_motor_power_loss:=maskbitFunction(Trip_BITs_16_to_31,14);
T_Emergency_stop:=maskbitFunction(Trip_BITs_16_to_31,15);
T_Sensor_failure_AI_276:=maskbitFunction(Trip_BITs_32_to_47,0);
T_Sensor_failure_AI_278:=maskbitFunction(Trip_BITs_32_to_47,1);
T_Sensor_failure_AI_280:=maskbitFunction(Trip_BITs_32_to_47,2);
T_Sensor_failure_AI_282:=maskbitFunction(Trip_BITs_32_to_47,3);
T_Sensor_failure_AI_288:=maskbitFunction(Trip_BITs_32_to_47,4);
T_Sensor_failure_AI_292:=maskbitFunction(Trip_BITs_32_to_47,5);
T_Sensor_failure_AI_272:=maskbitFunction(Trip_BITs_32_to_47,6);
T_Sensor_failure_AI_130:=maskbitFunction(Trip_BITs_32_to_47,7);
T_Sensor_failure_AI_134:=maskbitFunction(Trip_BITs_32_to_47,8);
T_Sensor_failure_AI_128:=maskbitFunction(Trip_BITs_32_to_47,9);
T_Sensor_failure_AI_256:=maskbitFunction(Trip_BITs_32_to_47,10);
T_Sensor_failure_AI_274:=maskbitFunction(Trip_BITs_32_to_47,11);
T_Sensor_failure_AI_270:=maskbitFunction(Trip_BITs_32_to_47,12);
T_Sensor_failure_AI_268:=maskbitFunction(Trip_BITs_32_to_47,13);
T_Sensor_failure_AI_286:=maskbitFunction(Trip_BITs_32_to_47,14);
T_Sensor_failure_AI_284:=maskbitFunction(Trip_BITs_32_to_47,15);
T_Sensor_failure_AI_304:=maskbitFunction(Trip_BITs_48_to_63,0);
T_Sensor_failure_AI_308:=maskbitFunction(Trip_BITs_48_to_63,1);
T_Sensor_failure_AI_312:=maskbitFunction(Trip_BITs_48_to_63,2);
T_Sensor_failure_AI_296:=maskbitFunction(Trip_BITs_48_to_63,3);
T_Sensor_failure_AI_300:=maskbitFunction(Trip_BITs_48_to_63,4);
T_Sensor_failure_AI_316:=maskbitFunction(Trip_BITs_48_to_63,5);
T_Sensor_failure_AI_262:=maskbitFunction(Trip_BITs_48_to_63,6);
T_Sensor_failure_AI_352:=maskbitFunction(Trip_BITs_48_to_63,7);
T_Sensor_failure_AI_354:=maskbitFunction(Trip_BITs_48_to_63,8);
T_Sensor_failure_AI_360:=maskbitFunction(Trip_BITs_48_to_63,9);
T_Sensor_failure_AI_362:=maskbitFunction(Trip_BITs_48_to_63,10);
T_Sensor_failure_AI_364:=maskbitFunction(Trip_BITs_48_to_63,11);
T_Rotating_stall_trip:=maskbitFunction(Trip_BITs_48_to_63,12);
T_Analog_inputs:=maskbitFunction(Trip_BITs_48_to_63,13);
T_High_oil_filter_diff_press:=maskbitFunction(Trip_BITs_48_to_63,14);
T_Sensor_failure_AI_260:=maskbitFunction(Trip_BITs_48_to_63,15);
A_High_comp_motor_winding_temp:=maskbitFunction(Trip_BITs_64_to_79,0);
A_High_comp_mo_DE_bear_temp:=maskbitFunction(Trip_BITs_64_to_79,1);
A_High_comp_mo_NDE_bear_temp:=maskbitFunction(Trip_BITs_64_to_79,2);
A_High_motor_air_temp:=maskbitFunction(Trip_BITs_64_to_79,3);
A_Low_chilled_medium_flow:=maskbitFunction(Trip_BITs_64_to_79,4);
A_High_chilled_medium_flow:=maskbitFunction(Trip_BITs_64_to_79,5);
A_Low_sea_water_flow:=maskbitFunction(Trip_BITs_64_to_79,6);
A_High_condenser_flow:=maskbitFunction(Trip_BITs_64_to_79,7);
T_Sensor_failure_AI_258:=maskbitFunction(Trip_BITs_64_to_79,8);
T_Sensor_failure_AI_264:=maskbitFunction(Trip_BITs_64_to_79,9);
T_Sensor_failure_AI_266:=maskbitFunction(Trip_BITs_64_to_79,10);
A_Rotating_stall:=maskbitFunction(Trip_BITs_64_to_79,11);
A_Low_oil_diff_pressure:=maskbitFunction(Trip_BITs_64_to_79,12);
A_High_oil_filter_diff_press:=maskbitFunction(Trip_BITs_64_to_79,13);
A_High_control_panel_temp:=maskbitFunction(Trip_BITs_64_to_79,14);
//A_Spare:=maskbitFunction(Trip_BITs_64_to_79,15);
Unit_running:=maskbitFunction(Status_BITs_0_to_15,0);
Unit_available:=maskbitFunction(Status_BITs_0_to_15,1);
Unit_remote:=maskbitFunction(Status_BITs_0_to_15,2);
Unit_auto:=maskbitFunction(Status_BITs_0_to_15,3);
Anti_recycle_status:=maskbitFunction(Status_BITs_0_to_15,4);
//S_Spare:=maskbitFunction(Status_BITs_0_to_15,5);
//S_Spare:=maskbitFunction(Status_BITs_0_to_15,6);
//S_Spare:=maskbitFunction(Status_BITs_0_to_15,7);
//S_Spare:=maskbitFunction(Status_BITs_0_to_15,8);
Unit_trip:=maskbitFunction(Status_BITs_0_to_15,9);
Unit_alarm:=maskbitFunction(Status_BITs_0_to_15,10);
Unit_fault:=maskbitFunction(Status_BITs_0_to_15,11);
Power_available:=maskbitFunction(Status_BITs_0_to_15,12);
Power_request:=maskbitFunction(Status_BITs_0_to_15,13);
//S_Spare:=maskbitFunction(Status_BITs_0_to_15,14);
PrV_in_min:=maskbitFunction(Status_BITs_0_to_15,15);
Unit_manual:=maskbitFunction(Status_BITs_16_to_31,0);
T_High_temp_oil_inlet_comp:=maskbitFunction(Status_BITs_16_to_31,1);
Unit_start_switch:=maskbitFunction(Status_BITs_16_to_31,2);
Sea_water_pump:=maskbitFunction(Status_BITs_16_to_31,3);

// Graphic controls
IF Unit_remote THEN
	Unit_switch_status:=2;
ELSIF Unit_auto THEN 
	Unit_switch_status:=3;
ELSIF Unit_manual THEN 
	Unit_switch_status:=4;

END_IF ;	

IF select_trendvalue > 0 THEN
	show_trendvalue[select_trendvalue]:= TRUE;
ELSIF select_trendvalue = 0 THEN
	FOR i := 0 TO 50 DO
      show_trendvalue[i] := FALSE;
   	END_FOR
END_IF ;	
	
// timer2 (IN:= TRUE, PT:=T#5S);;
//	IF timer2_Q THEN
//		Temp_motor_bearing_DE := Temp_motor_bearing_DE +1;
//		Motor_current := Motor_current + 1 ;
//		Timer2(IN:= FALSE);
//	END_IF

END_PROGRAM

// Chiller_1
PROGRAM Chiller_1
VAR

timer2 : standard.ton ;
{attribute 'ac_datalog_set_default_group' := 'DatalogChannel_1'}
instStruct : LogStruct;

modbus_var : ARRAY[0..100] OF INT;
modbus_var_1000 : ARRAY[0..123] OF WORD;
modbus_var_1001 : ARRAY[124..247] OF WORD;
modbus_var_1002 : ARRAY[248..371] OF WORD;
{attribute 'ac_datalog_hysteresis' := '0.2'}
{attribute 'ac_datalog' := 'DatalogChannel_1'}
Temp_chilled_medium_out : REAL;
{attribute 'ac_datalog_hysteresis' := '0.2'}
{attribute 'ac_datalog' := 'DatalogChannel_1'}
Temp_chilled_medium_in : REAL;
{attribute 'ac_datalog_hysteresis' := '0.2'}
{attribute 'ac_datalog' := 'DatalogChannel_1'}
Temp_water_inlet_cond : REAL;
{attribute 'ac_datalog_hysteresis' := '0.2'}
{attribute 'ac_datalog' := 'DatalogChannel_1'}
Press_suction_compr : REAL;
{attribute 'ac_datalog_hysteresis' := '0.5'}
{attribute 'ac_datalog' := 'DatalogChannel_1'}
Press_discharge_compr : REAL;
{attribute 'ac_datalog_hysteresis' := '0.5'}
{attribute 'ac_datalog' := 'DatalogChannel_1'}
Press_oil_receiver : REAL;
{attribute 'ac_datalog_hysteresis' := '0.5'}
{attribute 'ac_datalog' := 'DatalogChannel_1'}
Press_oil_compr : REAL;
{attribute 'ac_datalog_hysteresis' := '0.4'}
{attribute 'ac_datalog' := 'DatalogChannel_1'}
Temp_discharge : REAL;
{attribute 'ac_datalog_hysteresis' := '0.5'}
{attribute 'ac_datalog' := 'DatalogChannel_1'}
Oil_temp_receiver : REAL;
{attribute 'ac_datalog_hysteresis' := '0.5'}
{attribute 'ac_datalog' := 'DatalogChannel_1'}
Max_motor_temp : REAL;
{attribute 'ac_datalog_hysteresis' := '0.2'}
{attribute 'ac_datalog' := 'DatalogChannel_1'}
Temp_motor_bearing_DE : REAL;
{attribute 'ac_datalog_hysteresis' := '0.2'}
{attribute 'ac_datalog' := 'DatalogChannel_1'}
Temp_motor_bearing_NDE : REAL;
{attribute 'ac_datalog_hysteresis' := '4'}
{attribute 'ac_datalog' := 'DatalogChannel_1'}
Motor_current : REAL;
{attribute 'ac_datalog_hysteresis' := '50'}
{attribute 'ac_datalog' := 'DatalogChannel_1'}
Running_hours_comp_unscaled : WORD;
{attribute 'ac_datalog_hysteresis' := '50'}
{attribute 'ac_datalog' := 'DatalogChannel_1'}
Running_hours_oil_pump_unscaled : WORD;
{attribute 'ac_datalog' := 'DatalogChannel_1'}
Anti_recycle_time : REAL;
{attribute 'ac_datalog_hysteresis' := '2'}
{attribute 'ac_datalog' := 'DatalogChannel_1'}
Feedback_compressor : REAL;
{attribute 'ac_datalog_hysteresis' := '0.2'}
{attribute 'ac_datalog' := 'DatalogChannel_1'}
Oil_diff_pressure : REAL;
{attribute 'ac_datalog_hysteresis' := '0.3'}
{attribute 'ac_datalog' := 'DatalogChannel_1'}
Suction_saturated_temp : REAL;
{attribute 'ac_datalog_hysteresis' := '0.2'}
{attribute 'ac_datalog' := 'DatalogChannel_1'}
Discharge_saturated_temp : REAL;
{attribute 'ac_datalog_hysteresis' := '0.2'}
{attribute 'ac_datalog' := 'DatalogChannel_1'}
Temp_water_outlet_cond : REAL;
{attribute 'ac_datalog_hysteresis' := '0.2'}
{attribute 'ac_datalog' := 'DatalogChannel_1'}
Temp_motor_wind_R : REAL;
{attribute 'ac_datalog_hysteresis' := '0.2'}
{attribute 'ac_datalog' := 'DatalogChannel_1'}
Temp_motor_wind_S : REAL;
{attribute 'ac_datalog_hysteresis' := '0.2'}
{attribute 'ac_datalog' := 'DatalogChannel_1'}
Temp_motor_wind_T : REAL;
{attribute 'ac_datalog_hysteresis' := '0.2'}
{attribute 'ac_datalog' := 'DatalogChannel_1'}
Temp_motor_air : REAL;
{attribute 'ac_datalog_hysteresis' := '0.04'}
{attribute 'ac_datalog' := 'DatalogChannel_1'}
dP_CW : REAL;
{attribute 'ac_datalog_hysteresis' := '0.04'}
{attribute 'ac_datalog' := 'DatalogChannel_1'}
dP_SW : REAL;
{attribute 'ac_datalog_hysteresis' := '4'}
{attribute 'ac_datalog' := 'DatalogChannel_1'}
Chiller_capacity : REAL;
{attribute 'ac_datalog_hysteresis' := '2'}
{attribute 'ac_datalog' := 'DatalogChannel_1'}
Temp_oil_inlet_compr : REAL;
Spare : REAL;
{attribute 'ac_datalog_hysteresis' := '2'}
{attribute 'ac_datalog' := 'DatalogChannel_1'}
SP_CW_controller : REAL;
{attribute 'ac_datalog_hysteresis' := '2'}
{attribute 'ac_datalog' := 'DatalogChannel_1'}
Setpoint_oil_pump : REAL;
{attribute 'ac_datalog_hysteresis' := '0.02'}
{attribute 'ac_datalog' := 'DatalogChannel_1'}
Thrust_bearing_position : REAL;
{attribute 'ac_datalog_hysteresis' := '50'}
{attribute 'ac_datalog' := 'DatalogChannel_1'}
Oil_pump_running_hours : REAL;
{attribute 'ac_datalog_hysteresis' := '5'}
{attribute 'ac_datalog' := 'DatalogChannel_1'}
Liquid_level_condenser : REAL;
{attribute 'ac_datalog_hysteresis' := '0.05'}
{attribute 'ac_datalog' := 'DatalogChannel_1'}
Oil_Filter_Drop : REAL; 
{attribute 'ac_datalog_hysteresis' := '2'}
{attribute 'ac_datalog' := 'DatalogChannel_1'}
Proximitor_thrust_pos : REAL;
{attribute 'ac_datalog_hysteresis' := '0.4'}
{attribute 'ac_datalog' := 'DatalogChannel_1'}
Press_chilled_medium_in : REAL;
{attribute 'ac_datalog_hysteresis' := '0.2'}
{attribute 'ac_datalog' := 'DatalogChannel_1'}
Press_water_cond_out : REAL;
{attribute 'ac_datalog_hysteresis' := '0.02'}
{attribute 'ac_datalog' := 'DatalogChannel_1'}
Feedback_sea_water_valve : REAL;
{attribute 'ac_datalog_hysteresis' := '1'}
{attribute 'ac_datalog' := 'DatalogChannel_1'}
Oil_pressure_before_filter : REAL;
{attribute 'ac_datalog_hysteresis' := '0.2'}
{attribute 'ac_datalog' := 'DatalogChannel_1'}
Trafo_winding_temp : REAL;
{attribute 'ac_datalog_hysteresis' := '1'}
{attribute 'ac_datalog' := 'DatalogChannel_1'}
Feedback_VGD : REAL;
{attribute 'ac_datalog_hysteresis' := '4'}
{attribute 'ac_datalog' := 'DatalogChannel_1'}
Feedback_liquid_valve : REAL;
{attribute 'ac_datalog_hysteresis' := '3'}
{attribute 'ac_datalog' := 'DatalogChannel_1'}
Feedback_HGV : REAL;
{attribute 'ac_datalog_hysteresis' := '2'}
{attribute 'ac_datalog' := 'DatalogChannel_1'}
Discharge_superheat : REAL;
{attribute 'ac_datalog_hysteresis' := '0.6'}
{attribute 'ac_datalog' := 'DatalogChannel_1'}
Frequency_oil_pump : REAL;
{attribute 'ac_datalog_hysteresis' := '3'}
{attribute 'ac_datalog' := 'DatalogChannel_1'}
Hot_gas_valve_output : REAL;
{attribute 'ac_datalog_hysteresis' := '2'}
{attribute 'ac_datalog' := 'DatalogChannel_1'}
Control_signal_unit_d : REAL;
{attribute 'ac_datalog_hysteresis' := '2'}
{attribute 'ac_datalog' := 'DatalogChannel_1'}
Stall_detector : REAL;
{attribute 'ac_datalog_hysteresis' := '0.2'}
{attribute 'ac_datalog' := 'DatalogChannel_1'}
SP_MC_controller : REAL;
{attribute 'ac_datalog_hysteresis' := '2'}
{attribute 'ac_datalog' := 'DatalogChannel_1'}
Prerotary_output : REAL;
{attribute 'ac_datalog_hysteresis' := '2'}
{attribute 'ac_datalog' := 'DatalogChannel_1'}
VGD_output : REAL;
{attribute 'ac_datalog_hysteresis' := '2'}
{attribute 'ac_datalog' := 'DatalogChannel_1'}
SP_PID_compressor : REAL;
{attribute 'ac_datalog_hysteresis' := '2'}
{attribute 'ac_datalog' := 'DatalogChannel_1'}
Output_PID_suction : REAL;
{attribute 'ac_datalog_hysteresis' := '2'}
{attribute 'ac_datalog' := 'DatalogChannel_1'}
Output_PID_discharge : REAL;
{attribute 'ac_datalog_hysteresis' := '2'}
{attribute 'ac_datalog' := 'DatalogChannel_1'}
Output_PID_motor : REAL;
{attribute 'ac_datalog_hysteresis' := '2'}
{attribute 'ac_datalog' := 'DatalogChannel_1'}
Output_PID_superheat : REAL;
{attribute 'ac_datalog_hysteresis' := '2'}
{attribute 'ac_datalog' := 'DatalogChannel_1'}
SP_control : REAL;
{attribute 'ac_datalog_hysteresis' := '2'}
{attribute 'ac_datalog' := 'DatalogChannel_1'}
Unit_control_signal : REAL;
{attribute 'ac_datalog_hysteresis' := '2'}
{attribute 'ac_datalog' := 'DatalogChannel_1'}
Feedback_PRV : REAL;
{attribute 'ac_datalog_hysteresis' := '0.3'}
{attribute 'ac_datalog' := 'DatalogChannel_1'}
Theta_out : REAL;
{attribute 'ac_datalog_hysteresis' := '50'}
{attribute 'ac_datalog' := 'DatalogChannel_1'}
Alarm_limit_stall_count_unscaled : WORD;
{attribute 'ac_datalog_hysteresis' := '50'}
{attribute 'ac_datalog' := 'DatalogChannel_1'}
Alarm_limit_stall_count : REAL;
{attribute 'ac_datalog_hysteresis' := '2'}
{attribute 'ac_datalog' := 'DatalogChannel_1'}
Stall_ramp : REAL;
Min_allowed_PRVposition : REAL;
Number_of_starts : REAL;
SP_freq_oil_pump_VFD : REAL;
SP_oil_pressure_diff : REAL;
SP_oil_pressure : REAL;
{attribute 'ac_datalog_hysteresis' := '2'}
{attribute 'ac_datalog' := 'DatalogChannel_1'}
Setpoint_conv_oil_pump : REAL;
Days_above_stall_limit : REAL;
Hrs_above_stall_limit : REAL;
Min_above_stall_limit : REAL;
Sec_above_stall_limit : REAL;
{attribute 'ac_datalog_hysteresis' := '2'}
{attribute 'ac_datalog' := 'DatalogChannel_1'}
SP_cond_press : REAL;
{attribute 'ac_datalog_hysteresis' := '2'}
{attribute 'ac_datalog' := 'DatalogChannel_1'}
SP_PID_Level : REAL;
{attribute 'ac_datalog_hysteresis' := '2'}
{attribute 'ac_datalog' := 'DatalogChannel_1'}
Control_signal_SW_valve : REAL;
{attribute 'ac_datalog_hysteresis' := '4'}
{attribute 'ac_datalog' := 'DatalogChannel_1'}
Liquid_valve_output : REAL;
{attribute 'ac_datalog_hysteresis' := '0.2'}
{attribute 'ac_datalog' := 'DatalogChannel_1'}
SP_PID_seawater : REAL;
{attribute 'ac_datalog_hysteresis' := '4'}
{attribute 'ac_datalog' := 'DatalogChannel_1'}
Chiller_capacity_t1 : REAL;
{attribute 'ac_datalog_hysteresis' := '2'}
{attribute 'ac_datalog' := 'DatalogChannel_1'}
SW_pump_speed_order : REAL;
{attribute 'ac_datalog_hysteresis' := '0.4'}
{attribute 'ac_datalog' := 'DatalogChannel_1'}
Press_chilled_medium_out : REAL;
{attribute 'ac_datalog_hysteresis' := '50'}
{attribute 'ac_datalog' := 'DatalogChannel_1'}
Running_hours_compressormotor : REAL;
{attribute 'ac_datalog_hysteresis' := '0.2'}
{attribute 'ac_datalog' := 'DatalogChannel_1'}
Press_water_cond_inlet : REAL;
{attribute 'ac_datalog_hysteresis' := '2'}
{attribute 'ac_datalog' := 'DatalogChannel_1'}
Speed_feedback_VFD : REAL;
{attribute 'ac_datalog_hysteresis' := '2'}
{attribute 'ac_datalog' := 'DatalogChannel_1'}
Order_VFD_perc : REAL;
{attribute 'ac_datalog_hysteresis' := '2'}
{attribute 'ac_datalog' := 'DatalogChannel_1'}
Order_VFD_Hz : REAL;
{attribute 'ac_datalog_hysteresis' := '2'}
{attribute 'ac_datalog' := 'DatalogChannel_1'}
Temp_trafo_wind_U : REAL;
{attribute 'ac_datalog_hysteresis' := '0.2'}
{attribute 'ac_datalog' := 'DatalogChannel_1'}
Temp_trafo_wind_V : REAL;
{attribute 'ac_datalog_hysteresis' := '0.2'}
{attribute 'ac_datalog' := 'DatalogChannel_1'}
Temp_trafo_wind_W : REAL;
{attribute 'ac_datalog_hysteresis' := '2'}
{attribute 'ac_datalog' := 'DatalogChannel_1'}
Opt_speed_VFD_perc : REAL;
{attribute 'ac_datalog_hysteresis' := '2'}
{attribute 'ac_datalog' := 'DatalogChannel_1'}
Opt_speed_VFD_Hz : REAL;
Surge_counter_VFD : REAL;
Spare_4 : REAL;
Spare_3 : REAL;
Spare_2 : REAL;
Spare_0 : REAL;
Vibration_compressor_DE: REAL;
Vibration_compressor_NDE: REAL;
Feedback_seawater_valve_overboard : REAL;
Feedback_seawater_valve_bypass : REAL;
CW_flow_m3: REAL;
SW_flow_m3: REAL;
Max_motor_wind_temp: REAL;
Order_SWW_overboard: REAL;
Order_SWW_bypass: REAL;
{attribute 'ac_datalog_hysteresis' := '0.4'}
{attribute 'ac_datalog' := 'DatalogChannel'}
COP_chiller_mech : REAL ;
{attribute 'ac_datalog_hysteresis' := '50'}
{attribute 'ac_datalog' := 'DatalogChannel'}
P2_mot_1_kW : REAL ;
{attribute 'ac_datalog_hysteresis' := '50'}
{attribute 'ac_datalog' := 'DatalogChannel'}
P1_motor_kW : REAL ;
{attribute 'ac_datalog_hysteresis' := '0.4'}
{attribute 'ac_datalog' := 'DatalogChannel'}
COP_chiller_ele : REAL ;
{attribute 'ac_datalog_hysteresis' := '0.2'}
{attribute 'ac_datalog' := 'DatalogChannel'}
PI_chiller : REAL ;
;{attribute 'ac_datalog_hysteresis' := '40'}
{attribute 'ac_datalog' := 'DatalogChannel'}
Wasted_energy_kW : REAL ;
{attribute 'ac_datalog_hysteresis' := '200'}
{attribute 'ac_datalog' := 'DatalogChannel'}
Chiller_capacity_kW : REAL;
Thrust_bearing_ref_min : REAL ;
Thrust_bearing_ref_max : REAL ;
Thrust_bearing_ref : REAL ;
Q2_chillerMWh : REAL ;
Chiller_P1_MWh : REAL ;
Cal_date_MMYY : REAL ;
Chiller_P2_MWh : REAL ;
Liquid_line_temp : REAL ;
VFD_motor_current : REAL ;
Feedback_liquid_valve_raw : REAL ;
Feedback_VGD_raw : REAL ;
Feedback_PRV_raw : REAL ;
Feedback_HGV_raw : REAL ;
Feedback_seawater_valve_overboard_raw : REAL ;
Feedback_seawater_valve_bypass_raw : REAL ;
SP_cond_press_limit : REAL ;
SP_evap_press_limit : REAL ;
SP_discharge_superheat_limit : REAL ;
SP_t1 : REAL ;
VFD_min_allowed_frequence : REAL ;
VFD_min_allowed_speed : REAL ;

Trip_BITs_0_to_15 : WORD;
Trip_BITs_16_to_31: WORD;
Trip_BITs_32_to_47: WORD;
Trip_BITs_48_to_63: WORD;
Trip_BITs_64_to_79: WORD;
Trip_BITs_80_to_95: WORD;
Trip_BITs_96_to_121: WORD;
Trip_BITs_122_to_137: WORD;
Trip_BITs_138_to_153: WORD;
Trip_BITs_154_to_169: WORD;
Trip_BITs_170_to_185: WORD;
Trip_BITs_186_to_201: WORD;


Alarm_BITs_0_to_15: WORD;
Alarm_BITs_16_to_31: WORD;
Alarm_BITs_32_to_47: WORD;
Alarm_BITs_48_to_63: WORD;
Alarm_BITs_64_to_79: WORD;
Alarm_BITs_80_to_95: WORD;
Alarm_BITs_96_to_111: WORD;

Status_BITs_0_to_15 : WORD;
Status_BITs_16_to_31 : WORD;
Status_BITs_32_to_47: WORD;
Status_BITs_48_to_63: WORD;
Status_BITs_64_to_79: WORD;
Status_BITs_80_to_95: WORD;
Status_BITs_96_to_111: WORD;
Status_BITs_112_to_127: WORD;




DI_Status_BITs_0_to_15 : WORD;
DI_Status_BITs_16_to_31: WORD;

DO_Status_BITs_16_to_31: WORD;
DO_Status_BITs_32_to_47: WORD;

T_Overload_compressor_motor : BOOL;
T_Compressor_running_failure : BOOL;
T_Low_chilled_medium_outlet : BOOL;
T_Low_sea_water_flow : BOOL;
T_Oil_level_motor_bearing : BOOL;

T_Low_oil_flow : BOOL;
T_Overload_oil_pump_motor : BOOL;
T_Oil_pump_running_failure : BOOL;
T_Low_oil_flow_trip : BOOL;
T_High_temp_oil_receiver : BOOL;
T_Low_temp_oil_receiver : BOOL;
T_Low_suction_pressure : BOOL;
T_High_suction_pressure : BOOL;
T_High_discharge_pressure : BOOL;
T_Low_discharge_pressure : BOOL;
T_High_discharge_temp : BOOL;
T_Low_oil_diff_pressure : BOOL;
T_High_diff_oil_pressure : BOOL;
T_Starting_to_long : BOOL;
T_Surge_detection : BOOL;
T_Comp_thrust_bearing_position : BOOL;
Spare_trip_1 : BOOL;
T_Chilled_pump_run_failure : BOOL;
T_Sea_water_pump_run_failure : BOOL;
T_Low_chilled_medium_flow : BOOL;
T_High_chilled_medium_flow : BOOL;
T_Low_condenser_flow : BOOL;
T_High_condenser_flow : BOOL;
T_Emergency_stop : BOOL;
T_High_comp_mot_DE_bear_temp : BOOL;
T_High_comp_mot_NDE_bear_temp : BOOL;
T_High_motor_air_temp : BOOL;
T_Comp_motor_leak_detection : BOOL;
T_High_comp_mot_DE_bear_vib : BOOL;
T_High_comp_mot_NDE_bear_Vib : BOOL;
T_High_comp_motor_wind_temp : BOOL;
Spare_trip_2 : BOOL;
T_Rotating_stall_trip : BOOL;
T_Analog_inputs : BOOL;
T_Feedback_CW_valve : BOOL;
T_Low_oil_diff_press_prelub : BOOL;
T_Low_oil_diff_press_standstil : BOOL;

T_Spare_3 : BOOL;
T_Spare_4 : BOOL;
T_Spare_5 : BOOL;
T_Spare_6 : BOOL;
T_Spare_7 : BOOL;
T_Spare_8 : BOOL;
T_High_temp_oil_inlet_comp : BOOL;
T_Comp_motor_power_loss : BOOL;
Spare_trip_3 : BOOL;
T_Cathodic_protect_sys_alarm : BOOL;
T_High_oil_filter_diff_press : BOOL;
T_Flow_switch_FT01 : BOOL;
T_Starter_failure_trip : BOOL;
T_Incorrect_feedback_starter_trip : BOOL;

A_VGD_fault : BOOL;
A_High_condenser_flow : BOOL;
A_Rotating_stall : BOOL;
A_High_temp_oil_inlet_comp : BOOL;
SpareAlarm_1 : BOOL;
A_High_motor_air_temp : BOOL;
A_High_control_panel_temp : BOOL;
A_Low_oil_diff_pressure : BOOL;
Spare_alarm_2 : BOOL;
A_High_comp_motor_winding_temp : BOOL;
A_High_comp_mo_DE_bear_temp : BOOL;
A_High_comp_mo_NDE_bear_temp : BOOL;
A_High_comp_mo_DE_bear_vib : BOOL;
A_High_comp_mo_NDE_bear_vib : BOOL;
A_Low_chilled_medium_flow : BOOL;
A_High_chilled_medium_flow : BOOL;
A_Low_sea_water_flow : BOOL;
A_Seawater_pump_not_running : BOOL;
A_Spare : BOOL;
A_Spare_1 : BOOL;
A_Spare_2 : BOOL;
A_Spare_3 : BOOL;
A_Spare_4 : BOOL;
A_Spare_5 : BOOL;
A_Spare_6 : BOOL;
A_Spare_7 : BOOL;
A_Spare_8 : BOOL;
A_Spare_9 : BOOL;
A_Spare_10 : BOOL;
A_Spare_11 : BOOL;
A_High_oil_filter_diff_press : BOOL;
A_Spare_12 : BOOL;
A_Spare_13 : BOOL;
A_Spare_14 : BOOL;
A_Spare_15 : BOOL;
A_Spare_16 : BOOL;
A_Spare_17 : BOOL;
Anti_recycle_status : BOOL;
Low_oil_temperature : BOOL;
Low_oil_temp_auto : BOOL;
Oil_heater : BOOL;
Sea_water_pump : BOOL;
Comp_oil_pump : BOOL;
Bearing_oil_pump : BOOL;
Solenoid_oil_return : BOOL;
Unit_running : BOOL;
Unit_remote : BOOL;
Unit_auto : BOOL;
Unit_manual : BOOL;
Unit_trip : BOOL;
Unit_alarm : BOOL;
Unit_fault : BOOL;
Unit_start_switch : BOOL;
Unit_available : BOOL;
S_Spare_1 : BOOL;
S_Spare_2 : BOOL;
S_Spare_3 : BOOL;
S_Spare_4 : BOOL;
S_Spare_5 : BOOL;
S_Spare_6 : BOOL;
S_Spare_7 : BOOL;
S_Spare_8 : BOOL;
Solenoid_liquid_inj: BOOL;
CW_Flow_ind : BOOL;
Open_chilled_water_valve : BOOL;
Feedback_chilled_water_valve : BOOL;
Open_order_swv_overboard : BOOL;
Close_order_swv_overboard : BOOL;
Open_order_swv_bypass : BOOL;
Close_order_swv_bypass : BOOL;
VFD_man_auto : BOOL ;
VFD_freq_jump_on : BOOL ;
VFD_ramp_100_perc : BOOL ;
VFD_locked_100_perc : BOOL;
VFD_ramp_d_PRVcontrol : BOOL;
PRV_control : BOOL;
VFD_control : BOOL;
VFD_fixed_speed : BOOL;
Spare_151: BOOL;
T_Transformer_winding_temp : BOOL;
A_Transformer_winding_temp : BOOL;
T_trafo_opening_main_breaker : BOOL;
T_VFD : BOOL;
VFD_ready : BOOL;
T_VFD_emergency_stop : BOOL;
T_Low_5VDC_supply : BOOL;
T_High_5VDC_supply : BOOL;
T_Spare_9 : BOOL;
T_Spare_10 : BOOL;
T_Spare_11 : BOOL;
T_Spare_12 : BOOL;
T_Spare_13 : BOOL;
T_Low_liquid_level : BOOL;
T_SW_pump_off_to_long : BOOL;
T_Softstarter_failure : BOOL;
T_Motorstarter_failure : BOOL ;
T_CW_valveopen_failure : BOOL ;
T_SW_valveopen_failure : BOOL ;
T_High_disch_superheat :BOOL ;
T_Low_disch_superheat :BOOL ;
T_High_CW_outlet_temp : BOOL;
T_Low_CW_outlet_temp : BOOL;
T_Low_CW_inlet_temp : BOOL;
T_High_CW_inlet_temp : BOOL;
T_High_SW_outlet_temp : BOOL;
T_Low_SW_outlet_temp : BOOL;
T_Low_SW_inlet_temp : BOOL;
T_High_SW_inlet_temp : BOOL;
T_High_motor_wind_temp_R : BOOL;
T_High_motor_wind_temp_S : BOOL;
T_High_motor_wind_temp_T : BOOL;
T_High_press_ratio : BOOL;
T_Low_press_ratio : BOOL;
T_Low_CW_dP : BOOL;
T_High_CW_dP : BOOL;
T_Low_SW_dP : BOOL;
T_High_SW_dP : BOOL;
T_Long_time_PRV : BOOL;
T_Comp_thrust_neg_move : BOOL;
T_Comp_thrust_pos_move : BOOL;
T_VGD_fault : BOOL;
T_Low_oilpress_prelube : BOOL;
T_Low_temp_oil_inlet_comp : BOOL;
T_Low_oilpress_standby : BOOL;
T_Rotating_stall : BOOL;

T_Sensor_failure_AI_128: BOOL;
T_Sensor_failure_AI_130: BOOL;
T_Sensor_failure_AI_134: BOOL;
T_Sensor_failure_AI_256: BOOL;
T_Sensor_failure_AI_258: BOOL;
T_Sensor_failure_AI_260: BOOL;
T_Sensor_failure_AI_262: BOOL;
T_Sensor_failure_AI_264: BOOL;
T_Sensor_failure_AI_266: BOOL;
T_Sensor_failure_AI_268: BOOL;
T_Sensor_failure_AI_270: BOOL;
T_Sensor_failure_AI_272: BOOL;
T_Sensor_failure_AI_274: BOOL;
T_Sensor_failure_AI_276: BOOL;
T_Sensor_failure_AI_278: BOOL;
T_Sensor_failure_AI_280: BOOL;
T_Sensor_failure_AI_282: BOOL;
T_Sensor_failure_AI_284: BOOL;
T_Sensor_failure_AI_286: BOOL;
T_Sensor_failure_AI_288: BOOL;
T_Sensor_failure_AI_290: BOOL;
T_Sensor_failure_AI_292: BOOL;
T_Sensor_failure_AI_294: BOOL;
T_Sensor_failure_AI_296: BOOL;
T_Sensor_failure_AI_298: BOOL;
T_Sensor_failure_AI_330: BOOL;
T_Sensor_failure_AI_320: BOOL;
T_Sensor_failure_AI_322: BOOL;
T_Sensor_failure_AI_324: BOOL;
T_Sensor_failure_AI_326: BOOL;
T_Sensor_failure_AI_328: BOOL;
T_Sensor_failure_AI_332: BOOL;
T_Sensor_failure_AI_334: BOOL;
T_Sensor_failure_AI_300: BOOL;
T_Sensor_failure_AI_302: BOOL;
T_Sensor_failure_AI_304: BOOL;
T_Sensor_failure_AI_306: BOOL;
T_Sensor_failure_AI_308: BOOL;
T_Sensor_failure_AI_310: BOOL;
T_Sensor_failure_AI_312: BOOL;
T_Sensor_failure_AI_314: BOOL;
T_Sensor_failure_AI_316: BOOL;
T_Sensor_failure_AI_318: BOOL;
T_Sensor_failure_AI_354: BOOL;
T_Sensor_failure_AI_360: BOOL;
T_Sensor_failure_AI_362: BOOL;
T_Sensor_failure_AI_368: BOOL;
T_Sensor_failure_AI_370: BOOL;
T_Sensor_failure_AI_372: BOOL;
T_Sensor_failure_AI_374: BOOL;
T_Sensor_failure_AI_376: BOOL;
T_Sensor_failure_AI_378: BOOL;
T_Sensor_failure_AI_380: BOOL;
T_Sensor_failure_AI_382: BOOL;
T_Sensor_failure_AI_336: BOOL;
T_Sensor_failure_AI_338: BOOL;
T_Sensor_failure_AI_340: BOOL;
T_Sensor_failure_AI_342: BOOL;
T_Sensor_failure_AI_344: BOOL;
T_Sensor_failure_AI_346: BOOL;
T_Sensor_failure_AI_348: BOOL;
T_Sensor_failure_AI_350: BOOL;
T_Sensor_failure_AI_752: BOOL;
T_Sensor_failure_AI_754: BOOL;
T_Sensor_failure_AI_756: BOOL;
T_Sensor_failure_AI_760: BOOL;
T_Sensor_failure_AI_772: BOOL;
T_Sensor_failure_AI_774: BOOL;
T_Sensor_failure_AI_776: BOOL;
T_Sensor_failure_AI_778: BOOL;
T_Sensor_failure_AI_780: BOOL;

A_high_disch_press : BOOL ;
A_low_disch_press : BOOL ;
A_Low_suction_pressure : BOOL;
A_High_suction_pressure : BOOL;
A_High_discharge_temp : BOOL;
A_High_oil_temp_receiver : BOOL;
A_Low_oil_temp_receiver : BOOL;
A_Low_temp_oil_inlet_comp : BOOL;
A_High_oil_diff_pressure : BOOL;
A_Low_discharge_superheat : BOOL;
A_High_discharge_superheat : BOOL;
A_Low_CW_outlet_temp : BOOL;
A_High_CW_outlet_temp : BOOL;
A_Low_CW_inlet_temp : BOOL;
A_High_CW_inlet_temp : BOOL;
A_High_SW_outlet_temp : BOOL;
A_Low_condenser_flow : BOOL;
A_High_press_ratio : BOOL;
A_Low_press_ratio : BOOL;
A_Motor_speed_low : BOOL;
A_Low_SW_outlet_temp : BOOL;
A_Low_SW_inlet_temp : BOOL;
A_High_SW_inlet_temp : BOOL;
A_High_suction_superheat : BOOL;
A_Low_suction_superheat : BOOL;
A_High_temp_oil_separator : BOOL;
A_Low_temp_oil_separator : BOOL;
A_High_motor_wind_temp_R : BOOL;
A_High_motor_wind_temp_S : BOOL;
A_High_motor_wind_temp_T : BOOL;
A_High_CW_dP : BOOL;
A_Low_CW_dP : BOOL;
A_High_SW_dP : BOOL;
A_Low_SW_dP : BOOL;

Start_inhib_time_between_Start : BOOL;
Start_inhib_time_beetween_Stop : BOOL;
Start_inhib_PRV_not_min : BOOL;
Start_inhib_Motor_overload : BOOL;
Remote_bilge_pump_control : BOOL;
CW_pump_running : BOOL;
A_Low_liquid_level : BOOL;
A_Suction_press_limit : BOOL;
A_Discharge_press_limit : BOOL;
A_Discharge_superheat_limit : BOOL;
A_Motor_current_limit : BOOL;


DI_0_0_Emergency_stop : BOOL;
DI_0_0 : BOOL;
DI_0_1 : BOOL;
DI_0_2_Fault_reset : BOOL;
DI_0_2 : BOOL;
DI_0_3 : BOOL;
DI_0_4 : BOOL;
DI_0_5 : BOOL;
DI_0_6_Overload_protection : BOOL;
DI_0_6 : BOOL;
DI_0_7 : BOOL;
DI_1_0_Overload_oilpump : BOOL;
DI_1_0 : BOOL;
DI_1_1 : BOOL;
DI_1_2 : BOOL;
DI_1_3 : BOOL;
Power_available : BOOL;
DI_1_4 : BOOL;
DI_1_5_Starter_failure : BOOL;
DI_1_5 : BOOL;
DI_8_0_Controlpanel_temp : BOOL;
DI_8_0 : BOOL;
DI_8_1 : BOOL;
DI_8_2_VGD_limit_switch : BOOL;
DI_8_2 : BOOL;
DI_8_3_water_leak_motor  : BOOL;
DI_8_3 : BOOL;
DI_8_4_Catodic_protection : BOOL;
DI_8_4 : BOOL;
DI_8_5_Trust_bearing_probe : BOOL;
DI_8_5 : BOOL;
DI_8_6_ESD_operation : BOOL;
DI_8_6 : BOOL;
DI_8_7 : BOOL;
DI_9_0_MV_breaker_available : BOOL;
DI_9_0 : BOOL;
DI_9_1 : BOOL;
DI_9_2_Safe_return_to_port : BOOL;
DI_9_2 : BOOL;
DI_9_3 : BOOL;
DI_9_4_VFD_emergency_stop : BOOL;
DI_9_4 : BOOL;
DI_9_5 : BOOL;
DI_9_6 : BOOL;
DI_9_7 : BOOL;
DO_0_0_Start_signal_comp : BOOL;
DO_0_0 : BOOL;
DO_0_1_Start_signal_oil_pump : BOOL;
DO_0_1 : BOOL;
DO_0_2_Start_signal_SW_pump : BOOL;
DO_0_2 : BOOL;
DO_0_3_Start_signal_CW_pump : BOOL;
DO_0_3 : BOOL;
DO_0_4_Solenoid_valve_oil : BOOL;
DO_0_4 : BOOL;
DO_0_5_Solenoid_valve_liquid : BOOL;
DO_0_5 : BOOL;
DO_0_6_Oil_heater : BOOL;
DO_0_6 : BOOL;
DO_0_7_Comp_heater : BOOL;
DO_0_7 : BOOL;
DO_1_0 : BOOL;
DO_1_1 : BOOL;
DO_8_0_Liquid_valve_open : BOOL;
DO_8_0 : BOOL;
DO_8_1_Liquid_valve_close : BOOL;
DO_8_1 : BOOL;
DO_8_2_VGD_open : BOOL;
DO_8_2 : BOOL;
DO_8_3_VGD_close : BOOL;
DO_8_3 : BOOL;
DO_8_4_PRV_open : BOOL;
DO_8_4 : BOOL;
DO_8_5_PRV_close : BOOL;
DO_8_5 : BOOL;
DO_8_6_HGV_open : BOOL;
DO_8_6 : BOOL;
DO_8_7_HGV_close : BOOL;
DO_8_7 : BOOL;
DO_9_0_Open_order_swv_overboard : BOOL;
DO_9_0 : BOOL;
DO_9_1_Close_order_swv_overboard : BOOL;
DO_9_1 : BOOL;
DO_9_2_Open_order_swv_bypass : BOOL;
DO_9_2 : BOOL;
DO_9_3_Close_order_swv_bypass : BOOL;
DO_9_3 : BOOL;
DO_9_4 : BOOL;
DO_9_5 : BOOL;
DO_9_6 : BOOL;
DO_9_7 : BOOL;
Power_request : BOOL;
DO_12_0 : BOOL;
DO_12_1_Compressor_ready : BOOL;
DO_12_1 : BOOL;
DO_12_2 : BOOL;
DO_12_3 : BOOL;
DO_12_4_Control_panel_alarm : BOOL;
DO_12_4 : BOOL;
DO_12_5_Auto_reset : BOOL;
DO_12_5 : BOOL;
DO_12_6_Unit_running : BOOL;
DO_12_6 : BOOL;
DO_12_7 : BOOL;
Start_inhib_time_Oil_receiver_temp : BOOL;
PrV_in_min : BOOL;



//Graphic variables
Unit_switch_status : INT;
i : INT;
show_trendvalue : ARRAY[0..50] OF BOOL;
select_trendvalue : INT :=0 ;

END_VAR

Temp_chilled_medium_out:=scaleFunction(modbus_var_1000[10],0.1, 0);
Temp_chilled_medium_in:=scaleFunction(modbus_var_1000[11],0.1, 0);
Temp_water_inlet_cond:=scaleFunction(modbus_var_1000[12],0.1, 0);
Press_suction_compr:=scaleFunction(modbus_var_1000[13],0.01, 0);
Press_discharge_compr:=scaleFunction(modbus_var_1000[14],0.01, 0);
Press_oil_receiver:=scaleFunction(modbus_var_1000[15],0.01, 0);
Press_oil_compr:=scaleFunction(modbus_var_1000[16],0.01, 0);
Temp_discharge:=scaleFunction(modbus_var_1000[17],0.1, 0);
Oil_temp_receiver:=scaleFunction(modbus_var_1000[18],0.1, 0);
Max_motor_temp:=scaleFunction(modbus_var_1000[19],0.1, 0);
Temp_motor_bearing_DE:=scaleFunction(modbus_var_1000[20],0.1, 0);
Temp_motor_bearing_NDE:=scaleFunction(modbus_var_1000[21],0.1, 0);
Motor_current:=scaleFunction(modbus_var_1000[22],1.0, 0);
Running_hours_comp_unscaled:=modbus_var_1000[23];
//Anti_recycle_time:=scaleFunction(modbus_var_1000[24],1.0, 0);
Feedback_compressor:=scaleFunction(modbus_var_1000[25],1.0, 0);
Oil_diff_pressure:=scaleFunction(modbus_var_1000[26],0.01, 0);
Suction_saturated_temp:=scaleFunction(modbus_var_1000[27],0.1, 0);
Discharge_saturated_temp:=scaleFunction(modbus_var_1000[28],0.1, 0);
Temp_water_outlet_cond:=scaleFunction(modbus_var_1000[29],0.1, 0);
Temp_motor_wind_R:=scaleFunction(modbus_var_1000[30],0.1, 0);
Temp_motor_wind_S:=scaleFunction(modbus_var_1000[31],0.1, 0);
Temp_motor_wind_T:=scaleFunction(modbus_var_1000[32],0.1, 0);
Temp_motor_air:=scaleFunction(modbus_var_1000[33],0.1, 0);
dP_CW:=scaleFunction(modbus_var_1000[34],0.01, 0);
dP_SW:=scaleFunction(modbus_var_1000[35],0.01, 0);
CW_flow_m3:=scaleFunction(modbus_var_1000[36],1.0, 0);
Temp_oil_inlet_compr:=scaleFunction(modbus_var_1000[37],0.1, 0);
//Stall_detector:=scaleFunction(modbus_var_1000[38],0.01, 0);
SP_CW_controller:=scaleFunction(modbus_var_1000[39],0.1, 0);
Feedback_sea_water_valve:=scaleFunction(modbus_var_1000[40],0.1, 0);
Oil_pressure_before_filter:=scaleFunction(modbus_var_1000[41],0.01, 0);
//Feedback_VGD:=scaleFunction(modbus_var_1000[42],0.1, 0);
Chiller_capacity:=scaleFunction(modbus_var_1000[43],0.1, 0);
Setpoint_oil_pump:=scaleFunction(modbus_var_1000[44],0.01, 0);
Thrust_bearing_position:=scaleFunction(modbus_var_1000[45],0.1, 0);
Oil_pump_running_hours:=scaleFunction(modbus_var_1000[46],10, 0);
Liquid_level_condenser:=scaleFunction(modbus_var_1000[47],0.1, 0);
Oil_Filter_Drop:=scaleFunction(modbus_var_1000[48],0.01, 0);
Proximitor_thrust_pos:=scaleFunction(modbus_var_1000[49],0.1, 0);
//Spare_old_write_bits:=scaleFunction(modbus_var_1000[50],1.0, 0);
Press_chilled_medium_in:=scaleFunction(modbus_var_1000[51],0.01, 0);
Press_water_cond_out:=scaleFunction(modbus_var_1000[52],0.01, 0);
Discharge_superheat:=scaleFunction(modbus_var_1000[53],0.1, 0);
Frequency_oil_pump:=scaleFunction(modbus_var_1000[54],0.1, 0);
Feedback_liquid_valve:=scaleFunction(modbus_var_1000[55],0.1, 0);
Hot_gas_valve_output:=scaleFunction(modbus_var_1000[56],0.1, 0);
Control_signal_unit_d:=scaleFunction(modbus_var_1000[57],0.1, 0);
SP_MC_controller:=scaleFunction(modbus_var_1000[58],0.1, 0);
Prerotary_output:=scaleFunction(modbus_var_1000[59],0.1, 0);
//VGD_output:=scaleFunction(modbus_var_1000[60],0.1, 0);
SP_PID_compressor:=scaleFunction(modbus_var_1000[61],0.1, 0);
Output_PID_suction:=scaleFunction(modbus_var_1000[62],0.1, 0);
Output_PID_discharge:=scaleFunction(modbus_var_1000[63],0.1, 0);
Output_PID_motor:=scaleFunction(modbus_var_1000[64],0.1, 0);
Output_PID_superheat:=scaleFunction(modbus_var_1000[65],0.1, 0);
SP_control:=scaleFunction(modbus_var_1000[66],0.1, 0);
Unit_control_signal:=scaleFunction(modbus_var_1000[67],0.1, 0);
Feedback_PRV:=scaleFunction(modbus_var_1000[68],0.1, 0);
Theta_out:=scaleFunction(modbus_var_1000[69],0.1, 0);
//Alarm_limit_stall_count:=scaleFunction(modbus_var_1000[70],1.0, 0);
//Stall_ramp:=scaleFunction(modbus_var_1000[71],0.1, 0);
//Min_allowed_PRVposition:=scaleFunction(modbus_var_1000[72],0.1, 0);
Number_of_starts:=scaleFunction(modbus_var_1000[73],1.0, 0);
SP_oil_pressure:=scaleFunction(modbus_var_1000[74],0.01, 0);
Setpoint_conv_oil_pump:=scaleFunction(modbus_var_1000[75],0.1, 0);
//Days_above_stall_limit:=scaleFunction(modbus_var_1000[76],1.0, 0);
//Hrs_above_stall_limit:=scaleFunction(modbus_var_1000[77],1.0, 0);
//Min_above_stall_limit:=scaleFunction(modbus_var_1000[78],1.0, 0);
//Sec_above_stall_limit:=scaleFunction(modbus_var_1000[79],1.0, 0);
SP_PID_Level:=scaleFunction(modbus_var_1000[80],0.1, 0);
Control_signal_SW_valve:=scaleFunction(modbus_var_1000[81],0.1, 0);
Feedback_HGV:=scaleFunction(modbus_var_1000[82],0.1, 0);
Liquid_valve_output:=scaleFunction(modbus_var_1000[83],0.1, 0);
SP_PID_seawater:=scaleFunction(modbus_var_1000[84],0.1, 0);
Chiller_capacity_t1:=scaleFunction(modbus_var_1000[85],0.1, 0);
SW_pump_speed_order:=scaleFunction(modbus_var_1000[86],0.1, 0);
Anti_recycle_time:=scaleFunction(modbus_var_1000[87],1.0, 0);
Press_chilled_medium_out:=scaleFunction(modbus_var_1000[88],0.01, 0);
Press_water_cond_inlet:=scaleFunction(modbus_var_1000[89],0.01, 0);
Running_hours_compressormotor:=scaleFunction(modbus_var_1000[90],10, 0);


Trip_BITs_0_to_15:=modbus_var_1000[0];
Trip_BITs_16_to_31:=modbus_var_1000[1];
Trip_BITs_32_to_47:=modbus_var_1000[2];
Trip_BITs_48_to_63:=modbus_var_1000[3];
Trip_BITs_64_to_79:=modbus_var_1000[4];
// Alarm_BITs_80_to_95:=modbus_var_1000[5];
// Alarm_BITs_96_to_111:=modbus_var_1000[6];
Status_BITs_0_to_15:=modbus_var_1000[5];
Status_BITs_16_to_31:=modbus_var_1000[6];


T_Low_suction_pressure:=maskbitFunction(Trip_BITs_0_to_15,0);
T_High_discharge_pressure:=maskbitFunction(Trip_BITs_0_to_15,1);
T_High_discharge_temp:=maskbitFunction(Trip_BITs_0_to_15,2);
T_Low_oil_diff_pressure:=maskbitFunction(Trip_BITs_0_to_15,3);
T_High_diff_oil_pressure:=maskbitFunction(Trip_BITs_0_to_15,4);
T_Starting_to_long:=maskbitFunction(Trip_BITs_0_to_15,5);
T_Surge_detection:=maskbitFunction(Trip_BITs_0_to_15,6);
T_Comp_thrust_bearing_position:=maskbitFunction(Trip_BITs_0_to_15,7);
T_Overload_compressor_motor:=maskbitFunction(Trip_BITs_0_to_15,8);
T_Compressor_running_failure:=maskbitFunction(Trip_BITs_0_to_15,9);
T_Low_chilled_medium_outlet:=maskbitFunction(Trip_BITs_0_to_15,10);
T_Low_oil_flow:=maskbitFunction(Trip_BITs_0_to_15,11);
T_Overload_oil_pump_motor:=maskbitFunction(Trip_BITs_0_to_15,12);
T_Oil_pump_running_failure:=maskbitFunction(Trip_BITs_0_to_15,13);
T_Low_oil_flow_trip:=maskbitFunction(Trip_BITs_0_to_15,14);
T_High_temp_oil_receiver:=maskbitFunction(Trip_BITs_0_to_15,15);
T_High_comp_motor_wind_temp:=maskbitFunction(Trip_BITs_16_to_31,0);
T_High_comp_mot_DE_bear_temp:=maskbitFunction(Trip_BITs_16_to_31,1);
T_High_comp_mot_NDE_bear_temp:=maskbitFunction(Trip_BITs_16_to_31,2);
T_High_motor_air_temp:=maskbitFunction(Trip_BITs_16_to_31,3);
T_Comp_motor_leak_detection:=maskbitFunction(Trip_BITs_16_to_31,4);
T_High_5VDC_supply:=maskbitFunction(Trip_BITs_16_to_31,5);
T_Low_5VDC_supply:=maskbitFunction(Trip_BITs_16_to_31,6);
T_Chilled_pump_run_failure:=maskbitFunction(Trip_BITs_16_to_31,7);
T_Sea_water_pump_run_failure:=maskbitFunction(Trip_BITs_16_to_31,8);
T_Low_chilled_medium_flow:=maskbitFunction(Trip_BITs_16_to_31,9);
T_High_chilled_medium_flow:=maskbitFunction(Trip_BITs_16_to_31,10);
T_Low_sea_water_flow:=maskbitFunction(Trip_BITs_16_to_31,11);
T_High_condenser_flow:=maskbitFunction(Trip_BITs_16_to_31,12);
A_High_temp_oil_inlet_comp:=maskbitFunction(Trip_BITs_16_to_31,13);
T_Comp_motor_power_loss:=maskbitFunction(Trip_BITs_16_to_31,14);
T_Emergency_stop:=maskbitFunction(Trip_BITs_16_to_31,15);
T_Sensor_failure_AI_276:=maskbitFunction(Trip_BITs_32_to_47,0);
T_Sensor_failure_AI_278:=maskbitFunction(Trip_BITs_32_to_47,1);
T_Sensor_failure_AI_280:=maskbitFunction(Trip_BITs_32_to_47,2);
T_Sensor_failure_AI_282:=maskbitFunction(Trip_BITs_32_to_47,3);
T_Sensor_failure_AI_288:=maskbitFunction(Trip_BITs_32_to_47,4);
T_Sensor_failure_AI_292:=maskbitFunction(Trip_BITs_32_to_47,5);
T_Sensor_failure_AI_272:=maskbitFunction(Trip_BITs_32_to_47,6);
T_Sensor_failure_AI_130:=maskbitFunction(Trip_BITs_32_to_47,7);
T_Sensor_failure_AI_134:=maskbitFunction(Trip_BITs_32_to_47,8);
T_Sensor_failure_AI_128:=maskbitFunction(Trip_BITs_32_to_47,9);
T_Sensor_failure_AI_256:=maskbitFunction(Trip_BITs_32_to_47,10);
T_Sensor_failure_AI_274:=maskbitFunction(Trip_BITs_32_to_47,11);
T_Sensor_failure_AI_270:=maskbitFunction(Trip_BITs_32_to_47,12);
T_Sensor_failure_AI_268:=maskbitFunction(Trip_BITs_32_to_47,13);
T_Sensor_failure_AI_286:=maskbitFunction(Trip_BITs_32_to_47,14);
T_Sensor_failure_AI_284:=maskbitFunction(Trip_BITs_32_to_47,15);
T_Sensor_failure_AI_304:=maskbitFunction(Trip_BITs_48_to_63,0);
T_Sensor_failure_AI_308:=maskbitFunction(Trip_BITs_48_to_63,1);
T_Sensor_failure_AI_312:=maskbitFunction(Trip_BITs_48_to_63,2);
T_Sensor_failure_AI_296:=maskbitFunction(Trip_BITs_48_to_63,3);
T_Sensor_failure_AI_300:=maskbitFunction(Trip_BITs_48_to_63,4);
T_Sensor_failure_AI_316:=maskbitFunction(Trip_BITs_48_to_63,5);
T_Sensor_failure_AI_262:=maskbitFunction(Trip_BITs_48_to_63,6);
//T_Sensor_failure_AI_352:=maskbitFunction(Trip_BITs_48_to_63,7);
T_Sensor_failure_AI_354:=maskbitFunction(Trip_BITs_48_to_63,8);
T_Sensor_failure_AI_360:=maskbitFunction(Trip_BITs_48_to_63,9);
T_Sensor_failure_AI_362:=maskbitFunction(Trip_BITs_48_to_63,10);
//T_Sensor_failure_AI_364:=maskbitFunction(Trip_BITs_48_to_63,11);
//T_Rotating_stall_trip:=maskbitFunction(Trip_BITs_48_to_63,12);
T_Analog_inputs:=maskbitFunction(Trip_BITs_48_to_63,13);
T_High_oil_filter_diff_press:=maskbitFunction(Trip_BITs_48_to_63,14);
T_Sensor_failure_AI_260:=maskbitFunction(Trip_BITs_48_to_63,15);
A_High_comp_motor_winding_temp:=maskbitFunction(Trip_BITs_64_to_79,0);
A_High_comp_mo_DE_bear_temp:=maskbitFunction(Trip_BITs_64_to_79,1);
A_High_comp_mo_NDE_bear_temp:=maskbitFunction(Trip_BITs_64_to_79,2);
A_High_motor_air_temp:=maskbitFunction(Trip_BITs_64_to_79,3);
A_Low_chilled_medium_flow:=maskbitFunction(Trip_BITs_64_to_79,4);
A_High_chilled_medium_flow:=maskbitFunction(Trip_BITs_64_to_79,5);
A_Low_sea_water_flow:=maskbitFunction(Trip_BITs_64_to_79,6);
A_High_condenser_flow:=maskbitFunction(Trip_BITs_64_to_79,7);
T_Sensor_failure_AI_258:=maskbitFunction(Trip_BITs_64_to_79,8);
T_Sensor_failure_AI_264:=maskbitFunction(Trip_BITs_64_to_79,9);
T_Sensor_failure_AI_266:=maskbitFunction(Trip_BITs_64_to_79,10);
A_Rotating_stall:=maskbitFunction(Trip_BITs_64_to_79,11);
A_Low_oil_diff_pressure:=maskbitFunction(Trip_BITs_64_to_79,12);
A_High_oil_filter_diff_press:=maskbitFunction(Trip_BITs_64_to_79,13);
A_High_control_panel_temp:=maskbitFunction(Trip_BITs_64_to_79,14);
//A_Spare:=maskbitFunction(Trip_BITs_64_to_79,15);
Unit_running:=maskbitFunction(Status_BITs_0_to_15,0);
Unit_available:=maskbitFunction(Status_BITs_0_to_15,1);
Unit_remote:=maskbitFunction(Status_BITs_0_to_15,2);
Unit_auto:=maskbitFunction(Status_BITs_0_to_15,3);
Anti_recycle_status:=maskbitFunction(Status_BITs_0_to_15,4);
//S_Spare:=maskbitFunction(Status_BITs_0_to_15,5);
//S_Spare:=maskbitFunction(Status_BITs_0_to_15,6);
//S_Spare:=maskbitFunction(Status_BITs_0_to_15,7);
//S_Spare:=maskbitFunction(Status_BITs_0_to_15,8);
Unit_trip:=maskbitFunction(Status_BITs_0_to_15,9);
Unit_alarm:=maskbitFunction(Status_BITs_0_to_15,10);
Unit_fault:=maskbitFunction(Status_BITs_0_to_15,11);
Power_available:=maskbitFunction(Status_BITs_0_to_15,12);
Power_request:=maskbitFunction(Status_BITs_0_to_15,13);
//S_Spare:=maskbitFunction(Status_BITs_0_to_15,14);
PrV_in_min:=maskbitFunction(Status_BITs_0_to_15,15);
Unit_manual:=maskbitFunction(Status_BITs_16_to_31,0);
T_High_temp_oil_inlet_comp:=maskbitFunction(Status_BITs_16_to_31,1);
Unit_start_switch:=maskbitFunction(Status_BITs_16_to_31,2);
Sea_water_pump:=maskbitFunction(Status_BITs_16_to_31,3);


// old values



// Graphic controls
IF Unit_remote THEN
	Unit_switch_status:=2;
ELSIF Unit_auto THEN 
	Unit_switch_status:=3;
ELSIF Unit_manual THEN 
	Unit_switch_status:=4;

END_IF ;	

IF select_trendvalue > 0 THEN
	show_trendvalue[select_trendvalue]:= TRUE;
ELSIF select_trendvalue = 0 THEN
	FOR i := 0 TO 50 DO
      show_trendvalue[i] := FALSE;
   	END_FOR
END_IF ;	
	
// timer2 (IN:= TRUE, PT:=T#5S);;
//	IF timer2_Q THEN
//		Temp_motor_bearing_DE := Temp_motor_bearing_DE +1;
//		Motor_current := Motor_current + 1 ;
//		Timer2(IN:= FALSE);
//	END_IF

END_PROGRAM

// Calculus
PROGRAM Calculus
VAR


// MWCC

NakW_chiller_3 : REAL ;
NakW_chiller_4 : REAL ;

COP_chiller_3 : REAL ;
COP_chiller_4 : REAL ;
NakW_chiller_5 : REAL ;
NakW_chiller_6 : REAL ;

COP_chiller_5 : REAL ;
COP_chiller_6 : REAL ;
{attribute 'ac_datalog_hysteresis' := '100'}
{attribute 'ac_datalog' := 'DatalogChannel'}
Tot_Power_motor : REAL ;
{attribute 'ac_datalog_hysteresis' := '300'}
{attribute 'ac_datalog' := 'DatalogChannel'}
Tot_Q2 : REAL ;
{attribute 'ac_datalog_hysteresis' := '100'}
{attribute 'ac_datalog' := 'DatalogChannel'}
Tot_Q2_MWh : REAL ;
{attribute 'ac_datalog_hysteresis' := '100'}
{attribute 'ac_datalog' := 'DatalogChannel'}
Tot_P1_MWh : REAL ;
Power_motor_3_kW : REAL ;
Power_motor_4_kW : REAL ;
Power_motor_5_kW : REAL ;
Power_motor_6_kW : REAL ;
Power_3_not_zero : REAL ;
Power_4_not_zero : REAL ;
Power_5_not_zero : REAL ;
Power_6_not_zero : REAL ;

// SE700
Q2kW_chiller_1 : REAL ;
Q2kW_chiller_2 : REAL ;
Chiller_1_dpCW_bar : REAL ;
Chiller_2_dpCW_bar : REAL ;
Chiller_1_SR_dpCW_bar : REAL ;
Chiller_2_SR_dpCW_bar : REAL ;
Power_motor_1_kW : REAL ;
Power_motor_2_kW : REAL ;
Power_1_not_zero : REAL ;
Power_2_not_zero : REAL ;
NakW_chiller_1 : REAL ;
NakW_chiller_2 : REAL ;
COP_chiller_1 : REAL ;
COP_chiller_2 : REAL ;



Power_3_not_zero_func: WORD := 100;
Power_4_not_zero_func :  WORD := 100;
COP_chiller_3_func :  WORD := 100;
COP_chiller_4_func :  WORD := 100;
Power_5_not_zero_func: WORD := 100;
Power_6_not_zero_func :  WORD := 100;
COP_chiller_5_func :  WORD := 100;
COP_chiller_6_func :  WORD := 100;
Tot_Power_motor_func :  WORD := 100;
Tot_Q2_func :  WORD := 100;
Tot_Q2_MWh_func :  WORD := 100;
Tot_Na_MWh_func :  WORD := 100;
Power_motor_3_kW_func :  WORD := 100;
Power_motor_4_kW_func :  WORD := 100;

// SE700

Man_Auto_Chiller_1_func :  WORD := 100;
Man_Auto_Chiller_2_func :  WORD := 100;
//SE700_Chiller_1_Modb|||VALISERR(LOCAL.MODBUS2.Chiller_1.Program_number);//
//SE700_Chiller_2_Modb|||VALISERR(LOCAL.MODBUS2.Chiller_2.Program_number);
Flow_factor_chiller1_func :  WORD := 100;
Flow_factor_chiller2_func :  WORD := 100;


SR_Nom_dP_bar_func :  WORD := 100;


Chiller_1_dT_func :  WORD := 100;
Chiller_2_dT_func :  WORD := 100;
Chiller_1_max_dT_func :  WORD := 100;
Chiller_2_max_dT_func :  WORD := 100;
Chiller_1_Capacity_func :  WORD := 100;
Chiller_2_Capacity_func :  WORD := 100;
Chiller_1_CapacitykW_func :  WORD := 100;
Chiller_2_CapacitykW_func :  WORD := 100;
Chiller_1_dpCW_bar_func :  WORD := 100;
Chiller_2_dpCW_bar_func :  WORD := 100;
Chiller_1_SR_dpCW_bar_func :  WORD := 100;
Chiller_2_SR_dpCW_bar_func :  WORD := 100;
Power_motor_1_kW_func :  WORD := 100;
Power_motor_2_kW_func :  WORD := 100;
Power_1_not_zero_func :  WORD := 100;
Power_2_not_zero_func :  WORD := 100;
COP_chiller_1_func :  WORD := 100;
COP_chiller_2_func :  WORD := 100;
Chiller_1_Capacity_corr_flow_factor_func :  WORD := 100;
Chiller_2_Capacity_corr_flow_factor_func :  WORD := 100;
// New Variables
PI_chiller_1  : REAL ;
PI_chiller_1_word : WORD ;
PI_Calc_Error_AC1 : BOOL ;
PI_chiller_2  : REAL ;
PI_chiller_2_word : WORD ;
PI_Calc_Error_AC2 : BOOL ;
PI_chiller_3  : REAL ;
PI_chiller_3_word : WORD ;
PI_Calc_Error_AC3 : BOOL ;
PI_chiller_4  : REAL ;
PI_chiller_4_word : WORD ;
PI_Calc_Error_AC4 : BOOL ;
PI_chiller_5  : REAL ;
PI_chiller_5_word : WORD ;
PI_Calc_Error_AC5 : BOOL ;
PI_chiller_6  : REAL ;
PI_chiller_6_word : WORD ;
PI_Calc_Error_AC6 : BOOL ;
delaytimer2 : TON ;	
resetbuttons : BOOL := FALSE  ;
COP_theo_AC1 :REAL ;	
COP_theo_AC2 :REAL ;
COP_theo_AC3 :REAL ;
COP_theo_AC4 :REAL ;
COP_theo_AC5 :REAL ;
COP_theo_AC6 :REAL ;
totRunningChillers : INT;
WastedEnergy_AC1 :REAL ;
WastedEnergy_AC1_word :WORD ;
WastedEnergy_AC2 :REAL ;
WastedEnergy_AC2_word :WORD ;
WastedEnergy_AC3 :REAL ;
WastedEnergy_AC3_word :WORD ;
WastedEnergy_AC4 :REAL ;
WastedEnergy_AC4_word :WORD ;
WastedEnergy_AC5 :REAL ;
WastedEnergy_AC5_word :WORD ;
WastedEnergy_AC6 :REAL ;
WastedEnergy_AC6_word :WORD ;
Total_PI : REAL ;
// Time variables
Result_time : SysTimeRtc.RTS_IEC_RESULT;
udiLocal_DateAndTime : UDINT;
current_date : UDINT ;

	
END_VAR

IF GVL.startUp THEN
	startupReadcsv();
	IF NOT GVL.startUp THEN	
		GVL.xReadCOP := FALSE;
		GVL.startdelaytimer :=TRUE;
	END_IF
	
END_IF

GVL.delaytimer (IN:= GVL.startdelaytimer, PT:=T#5S);
IF GVL.delaytimer.Q THEN
	GVL.xReadCOP := TRUE;
	GVL.startdelaytimer:=FALSE;
	resetbuttons := TRUE ;
END_IF
delaytimer2 (IN:= resetbuttons, PT:=T#5S);
IF delaytimer2.Q THEN
	GVL.xReadCOP := FALSE;
	GVL.initRead := FALSE;
	resetbuttons := FALSE;
END_IF

// Get system time
current_date := TO_UDINT(SysTimeRtcGet(Result_time));
Result_time := SysTimeRTCConvertUTCToLocal(current_date, udiLocal_DateAndTime);
GVL.CurrentDate := TO_DT(udiLocal_DateAndTime); // DT#2018-6-6-9:8:38

// MWCC
Tot_Q2_MWh:=Tot_Q2:=sequence.Chiller_1_Q2_MWh + sequence.Chiller_2_Q2_MWh + Sequence.Chiller_3_Q2_MWh + Sequence.Chiller_4_Q2_MWh;// + Sequence.Chiller_5_Q2_MWh + Sequence.Chiller_6_Q2_MWh ;
Tot_P1_MWh:=Tot_Q2:=sequence.Chiller_1_P1_MWh + sequence.Chiller_2_P1_MWh + Sequence.Chiller_3_P1_MWh + Sequence.Chiller_4_P1_MWh;// + Sequence.Chiller_5_P1_MWh + Sequence.Chiller_6_P1_MWh ;





//Power_1_not_zero:=Power_1_not_zero_func;
//Power_2_not_zero:=Power_2_not_zero_func;



// New Func
Power_motor_1_kW:=sequence.P1_motor_1_kW;
Power_motor_2_kW:=sequence.P1_motor_2_kW;
Power_motor_3_kW:=sequence.P1_motor_3_kW;
Power_motor_4_kW:=sequence.P1_motor_4_kW;
//Power_motor_5_kW:=sequence.P1_motor_5_kW;
//Power_motor_6_kW:=sequence.P1_motor_6_kW;

(*
NakW_chiller_1:=Power_not_zero_func(Power_motor_1_kW);
NakW_chiller_2:=Power_not_zero_func(Power_motor_2_kW);
NakW_chiller_3:=Power_not_zero_func(Power_motor_3_kW);
NakW_chiller_4:=Power_not_zero_func(Power_motor_4_kW);
*)
Tot_Power_motor:=Power_motor_1_kW + Power_motor_2_kW + Power_motor_3_kW + Power_motor_4_kW;// + Power_motor_5_kW +Power_motor_6_kW;
Tot_Q2:=sequence.Q2kW_chiller_1 + sequence.Q2kW_chiller_2 + Sequence.Q2kW_chiller_3 + Sequence.Q2kW_chiller_4;// + Sequence.Q2kW_chiller_5 + Sequence.Q2kW_chiller_6;

COP_chiller_1:=Sequence.COP_chiller_1_ele;
COP_chiller_2:=Sequence.COP_chiller_2_ele;
COP_chiller_3:=Sequence.COP_chiller_3_ele;
COP_chiller_4:=Sequence.COP_chiller_4_ele;
//COP_chiller_5:=Sequence.COP_chiller_5_ele;
//COP_chiller_6:=Sequence.COP_chiller_6_ele;

totRunningChillers := BOOL_TO_INT(Chiller_1.Unit_running) + BOOL_TO_INT(Chiller_2.Unit_running) + BOOL_TO_INT(Chiller_3.Unit_running) + BOOL_TO_INT(Chiller_4.Unit_running);// + BOOL_TO_INT(Chiller_5.Unit_running); // + BOOL_TO_INT(Chiller_6.Unit_running) ;

IF Chiller_1.Unit_running THEN
	PI_calculation(Chiller_1.Chiller_capacity,Chiller_1.Temp_water_inlet_cond,COP_chiller_1,Chiller_1.Temp_chilled_medium_out, 1, PI_act=>PI_chiller_1, noCalc_error=>PI_Calc_Error_AC1, COP_theo=>COP_theo_AC1);	
	WastedEnergy_AC1 := Wasted_calc(sequence.Q2kW_chiller_1, COP_theo_AC1, Power_motor_1_kW) ;
	ELSE
	PI_chiller_1 := 0;
	WastedEnergy_AC1 := 0;
	PI_Calc_Error_AC1 := TRUE;
	COP_theo_AC1 := 0;		
END_IF

IF Chiller_2.Unit_running THEN
	PI_calculation(Chiller_2.Chiller_capacity,Chiller_2.Temp_water_inlet_cond,COP_chiller_2,Chiller_2.Temp_chilled_medium_out, 2, PI_act=>PI_chiller_2,noCalc_error=>PI_Calc_Error_AC2, COP_theo=>COP_theo_AC2);
	WastedEnergy_AC2 := Wasted_calc(sequence.Q2kW_chiller_2, COP_theo_AC2, Power_motor_2_kW) ;
	ELSE
	PI_chiller_2 := 0;
	WastedEnergy_AC2 := 0;
	PI_Calc_Error_AC2 := TRUE ;
	COP_theo_AC2 := 0;		
END_IF

IF Chiller_3.Unit_running THEN
	PI_calculation(Chiller_3.Chiller_capacity,Chiller_3.Temp_water_inlet_cond,COP_chiller_3,Chiller_3.Temp_chilled_medium_out, 3, PI_act=>PI_chiller_3,noCalc_error=>PI_Calc_Error_AC3, COP_theo=>COP_theo_AC3);
	WastedEnergy_AC3 := Wasted_calc(sequence.Q2kW_chiller_3, COP_theo_AC3, Power_motor_3_kW) ;
	ELSE
	PI_chiller_3 := 0;
	WastedEnergy_AC3 := 0;	
	PI_Calc_Error_AC3 := TRUE ;
	COP_theo_AC3 := 0;		
END_IF

IF Chiller_4.Unit_running THEN
	PI_calculation(Chiller_4.Chiller_capacity,Chiller_4.Temp_water_inlet_cond,COP_chiller_4,Chiller_4.Temp_chilled_medium_out, 2, PI_act=>PI_chiller_4,noCalc_error=>PI_Calc_Error_AC4, COP_theo=>COP_theo_AC4);
	WastedEnergy_AC4 := Wasted_calc(sequence.Q2kW_chiller_4, COP_theo_AC4, Power_motor_4_kW) ;
	ELSE
	PI_chiller_4 := 0;
	WastedEnergy_AC4 := 0;
	PI_Calc_Error_AC4 := TRUE ;
	COP_theo_AC4 := 0;			
END_IF
(*
IF Chiller_5.Unit_running THEN
	PI_calculation(Chiller_5.Chiller_capacity,Chiller_5.Temp_water_inlet_cond,COP_chiller_5,Chiller_5.Temp_chilled_medium_out, 1, PI_act=>PI_chiller_5,noCalc_error=>PI_Calc_Error_AC5, COP_theo=>COP_theo_AC5);
	WastedEnergy_AC5 := Wasted_calc(sequence.Q2kW_chiller_5, COP_theo_AC5, Power_motor_5_kW) ;
	ELSE
	PI_chiller_5 := 0;
	WastedEnergy_AC5 := 0;
	PI_Calc_Error_AC5 := TRUE ;
	COP_theo_AC5 := 0;			
END_IF
*)


PI_chiller_1_word := REAL_TO_WORD(PI_chiller_1 * 100) ;
PI_chiller_2_word := REAL_TO_WORD(PI_chiller_2 * 100) ;
PI_chiller_3_word := REAL_TO_WORD(PI_chiller_3 * 100) ;
PI_chiller_4_word := REAL_TO_WORD(PI_chiller_4 * 100) ;
//PI_chiller_5_word := REAL_TO_WORD(PI_chiller_5 * 100) ;
//PI_chiller_6_word := REAL_TO_WORD(PI_chiller_6 * 100) ;

WastedEnergy_AC1_word := REAL_TO_WORD(WastedEnergy_AC1) ;
WastedEnergy_AC2_word := REAL_TO_WORD(WastedEnergy_AC2) ;
WastedEnergy_AC3_word := REAL_TO_WORD(WastedEnergy_AC3) ;
WastedEnergy_AC4_word := REAL_TO_WORD(WastedEnergy_AC4) ;
//WastedEnergy_AC5_word := REAL_TO_WORD(WastedEnergy_AC5) ;
//WastedEnergy_AC6_word := REAL_TO_WORD(WastedEnergy_AC6) ;

(*
PI_calculation(95,31,4.5,6.1, 1, PI_act=>PI_chiller_1 ,noCalc_error=>PI_Calc_Error_AC1, COP_theo=>COP_theo_AC1);
PI_calculation(92,31,4.5,6.1, 3, PI_act=>PI_chiller_2 ,noCalc_error=>PI_Calc_Error_AC2, COP_theo=>COP_theo_AC2);
PI_calculation(91,31,4.5,6.1, 2, PI_act=>PI_chiller_3 ,noCalc_error=>PI_Calc_Error_AC3, COP_theo=>COP_theo_AC3);
PI_calculation(90,31,4.5,6.1, 3, PI_act=>PI_chiller_4 ,noCalc_error=>PI_Calc_Error_AC4, COP_theo=>COP_theo_AC4);
*)

IF totRunningChillers>0 THEN
	Total_PI:=Tot_PI(PI_chiller_1, PI_chiller_2, PI_chiller_3, PI_chiller_4, PI_chiller_5, PI_chiller_6 , totRunningChillers) ; //
	ELSE 
	Total_PI := 0 ;
END_IF

END_PROGRAM

// AC_DataLogManager
//Code generated by Application Composer.
//Modifying generated code is not recommended!
FUNCTION_BLOCK AC_DataLogManager EXTENDS AC_DataLog.DataLogManager
VAR_INPUT 
    INST_DataLogChannel : AC_DataLogManager_DataLogChannel;
    INST_DataLogChannel_1 : AC_DataLogManager_DataLogChannel_1;
    INST_DataLogChannel_2 : AC_DataLogManager_DataLogChannel_2;
    INST_DataLogChannel_3 : AC_DataLogManager_DataLogChannel_3;
    INST_DataLogChannel_4 : AC_DataLogManager_DataLogChannel_4;
    AC_ARRAY_pitfDataLogChannels : ARRAY[0..4] OF AC_DataLog.IDataLogChannel;
END_VAR

//Code generated by Application Composer.
//Modifying generated code is not recommended!
SUPER^();

END_FUNCTION_BLOCK

// /AC_Plant_Overview
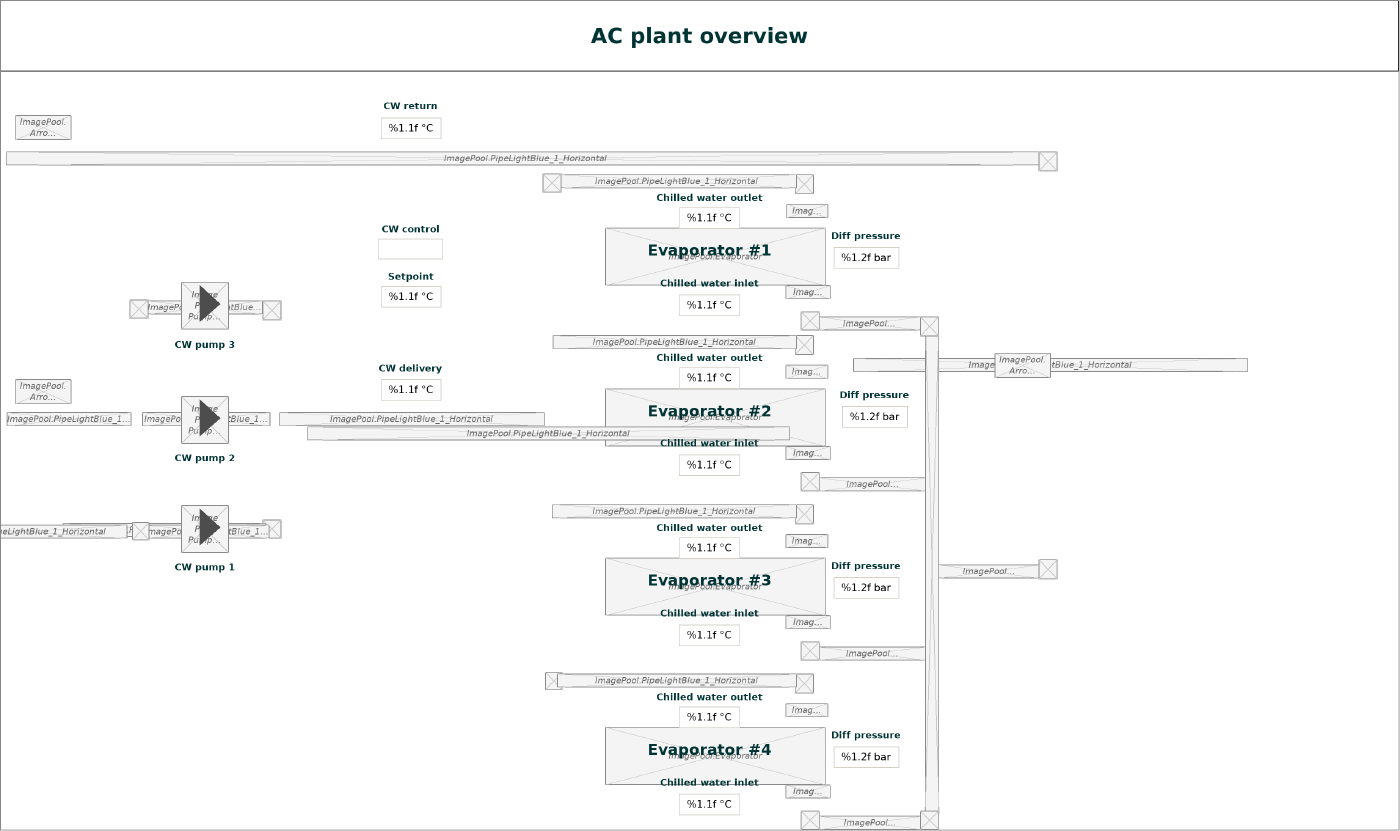
VISUALIZATION AC_Plant_Overview  // 1654x982
    Image (330,487 313x16), angle 180, image: ImagePool.PipeLightBlue_1_Horizontal
    Image (929,241 49x16), angle 90, image: ImagePool.PipeLightBlue_1_Horizontal
    Rectangle (0,0 1652x84)
    Label (295,7 1063x70), "AC plant overview"
    Image (7,179 1228x16), image: ImagePool.PipeLightBlue_1_Horizontal
    Image (1008,423 466x16), angle 90, image: ImagePool.PipeLightBlue_1_Horizontal
    Image (1108,667 121x16), angle 180, image: ImagePool.PipeLightBlue_1_Horizontal
    Image (1227,661 22x23), angle 180, image: ImagePool.PipeLightBlue_3_RD
    Image (966,374 122x16), image: ImagePool.PipeLightBlue_1_Horizontal
    Image (946,368 22x22), image: ImagePool.PipeLightBlue_3_RU
    Image (928,337 53x16), angle 270, image: ImagePool.PipeLightBlue_1_Horizontal
    Image (939,206 22x23), angle 90, image: ImagePool.PipeLightBlue_3_RD
    Image (715,269 260x68), image: ImagePool.Evaporator
    Label (761,276 155x40), "Evaporator #1"
    Image (658,206 283x16), image: ImagePool.PipeLightBlue_1_Horizontal
    Label (981,264 84x30), "Diff pressure"
    Textfield (985,292 77x25), "%1.2f bar", text variable: Chiller_1.dP_CW
        p4168582468: Chiller_1.dP_CW
    Textfield (802,348 72x25), "%1.1f °C", text variable: Chiller_1.Temp_chilled_medium_in
        p4168582468: Chiller_1.Temp_chilled_medium_in
    Label (778,323 121x24), "Chilled water inlet"
    Image (641,205 22x22), angle 90, image: ImagePool.PipeLightBlue_3_RU
    Image (644,794 20x21), angle 90, image: ImagePool.PipeLightBlue_2_LU
    Image (310,355 22x23), angle 90, image: ImagePool.PipeLightBlue_3_RD
    Image (310,614 22x22), angle 90, image: ImagePool.PipeLightBlue_1_LD
    Image (168,487 151x16), angle 180, image: ImagePool.PipeLightBlue_1_Horizontal
    Image (74,618 240x16), angle 90, image: ImagePool.PipeLightBlue_1_Horizontal
    Image (174,355 136x16), image: ImagePool.PipeLightBlue_1_Horizontal
    Image (171,620 147x16), image: ImagePool.PipeLightBlue_1_Horizontal
    Image (214,597 56x56), image: ImagePool.Pump_Large_3
    Image (214,468 56x56), image: ImagePool.Pump_Large_3
    Image (214,333 56x56), image: ImagePool.Pump_Large_3
    Image (153,354 22x22), angle 90, image: ImagePool.PipeLightBlue_3_RU
    Image (156,617 20x21), angle 90, image: ImagePool.PipeLightBlue_2_LU
    Image (8,487 147x16), angle 180, image: ImagePool.PipeLightBlue_1_Horizontal
    Image (18,136 66x29), angle 180, image: ImagePool.Arrow lightblue left
    Image (18,448 66x29), image: ImagePool.Arrow lightblue left
    Image (1175,417 66x29), angle 270, image: ImagePool.Arrow lightblue left
    Textfield (802,245 72x25), "%1.1f °C", text variable: Chiller_1.Temp_chilled_medium_out
        p4168582468: Chiller_1.Temp_chilled_medium_out
    Label (778,222 121x24), "Chilled water outlet"
    Image (928,431 50x16), angle 90, image: ImagePool.PipeLightBlue_1_Horizontal
    Image (966,564 130x16), image: ImagePool.PipeLightBlue_1_Horizontal
    Image (946,558 22x22), image: ImagePool.PipeLightBlue_3_RU
    Image (928,527 53x16), angle 270, image: ImagePool.PipeLightBlue_1_Horizontal
    Image (939,396 22x23), angle 90, image: ImagePool.PipeLightBlue_3_RD
    Image (715,459 260x68), image: ImagePool.Evaporator
    Label (761,466 155x40), "Evaporator #2"
    Image (653,396 288x16), image: ImagePool.PipeLightBlue_1_Horizontal
    Image (928,631 50x16), angle 90, image: ImagePool.PipeLightBlue_1_Horizontal
    Image (966,764 129x16), image: ImagePool.PipeLightBlue_1_Horizontal
    Image (946,758 22x22), image: ImagePool.PipeLightBlue_3_RU
    Image (928,727 53x16), angle 270, image: ImagePool.PipeLightBlue_1_Horizontal
    Image (939,596 22x23), angle 90, image: ImagePool.PipeLightBlue_3_RD
    Image (715,659 260x68), image: ImagePool.Evaporator
    Label (761,666 155x40), "Evaporator #3"
    Image (652,596 289x16), image: ImagePool.PipeLightBlue_1_Horizontal
    Label (981,654 84x30), "Diff pressure"
    Textfield (985,682 77x25), "%1.2f bar", text variable: Chiller_3.dP_CW
        p4168582468: Chiller_3.dP_CW
    Textfield (802,738 72x25), "%1.1f °C", text variable: Chiller_3.Temp_chilled_medium_in
        p4168582468: Chiller_3.Temp_chilled_medium_in
    Label (778,713 121x24), "Chilled water inlet"
    Textfield (802,635 72x25), "%1.1f °C", text variable: Chiller_3.Temp_chilled_medium_out
        p4168582468: Chiller_3.Temp_chilled_medium_out
    Label (778,612 121x24), "Chilled water outlet"
    Image (928,831 50x16), angle 90, image: ImagePool.PipeLightBlue_1_Horizontal
    Image (966,964 124x16), image: ImagePool.PipeLightBlue_1_Horizontal
    Image (946,958 22x22), image: ImagePool.PipeLightBlue_3_RU
    Image (928,927 53x16), angle 270, image: ImagePool.PipeLightBlue_1_Horizontal
    Image (939,796 22x23), angle 90, image: ImagePool.PipeLightBlue_3_RD
    Image (715,859 260x68), image: ImagePool.Evaporator
    Label (761,866 155x40), "Evaporator #4"
    Image (658,796 283x16), image: ImagePool.PipeLightBlue_1_Horizontal
    Label (981,854 84x30), "Diff pressure"
    Textfield (985,882 77x25), "%1.2f bar", text variable: Chiller_4.dP_CW
        p4168582468: Chiller_4.dP_CW
    Textfield (802,938 72x25), "%1.1f °C", text variable: Chiller_4.Temp_chilled_medium_in
        p4168582468: Chiller_4.Temp_chilled_medium_in
    Label (778,913 121x24), "Chilled water inlet"
    Textfield (802,835 72x25), "%1.1f °C", text variable: Chiller_4.Temp_chilled_medium_out
        p4168582468: Chiller_4.Temp_chilled_medium_out
    Label (778,812 121x24), "Chilled water outlet"
    Image (363,504 570x16), angle 90, image: ImagePool.PipeLightBlue_1_Horizontal
    Image (-93,620 243x16), angle 90, image: ImagePool.PipeLightBlue_1_Horizontal
    Label (454,315 63x24), "Setpoint"
    Textfield (450,338 71x25), "%1.1f °C", text variable: Sequence.Setpoint_CW
        p4168582468: Sequence.Setpoint_CW
    Image (1227,179 22x23), angle 90, image: ImagePool.PipeLightBlue_3_RD
    Image (1093,388 16x574), angle 180, image: ImagePool.PipeLightBlue_1_Vertical
    Image (1087,958 22x22), angle 90, image: ImagePool.PipeLightBlue_1_LD
    Image (1087,374 22x23), angle 90, image: ImagePool.PipeLightBlue_3_RD
    Textfield (450,139 71x25), "%1.1f °C", text variable: Sequence.Temp_inlet_chilled_water
        p4168582468: Sequence.Temp_inlet_chilled_water
    Textfield (450,448 71x25), "%1.1f °C", text variable: Sequence.Temp_outlet_chilled_water
        p4168582468: Sequence.Temp_outlet_chilled_water
    Label (438,422 94x27), "CW delivery"
    Textfield (447,282 76x24), tooltip "Sequence.CW_Control_inout", text variable: Sequence.CW_Control_inout, text list: 'TextList_in_outlet', text index: Sequence.CW_Control_inout
        OnMouseClick:  ToggleVariable=Sequence.Sequency_control
    Label (454,259 63x24), "CW control"
    Label (438,112 94x27), "CW return"
    Label (195,657 94x27), "CW pump 1"
    Label (195,528 94x27), "CW pump 2"
    Label (195,394 94x27), "CW pump 3"
    Polygon (236,356) (236,337) (260,359) (236,380) (236,372), colour toggle: Sequence.Chilled_medium_pump_3
    Polygon (236,491) (236,472) (260,494) (236,515) (236,507), colour toggle: Sequence.Chilled_medium_pump_2
    Polygon (236,620) (236,601) (260,623) (236,644) (236,636), colour toggle: Sequence.Chilled_medium_pump_1
    Label (991,452 84x30), "Diff pressure"
    Textfield (995,480 77x25), "%1.2f bar", text variable: Chiller_2.dP_CW
        p4168582468: Chiller_2.dP_CW
    Textfield (802,537 72x25), "%1.1f °C", text variable: Chiller_2.Temp_chilled_medium_in
        p4168582468: Chiller_2.Temp_chilled_medium_in
    Label (778,512 121x24), "Chilled water inlet"
    Textfield (802,434 72x25), "%1.1f °C", text variable: Chiller_2.Temp_chilled_medium_out
        p4168582468: Chiller_2.Temp_chilled_medium_out
    Label (778,411 121x24), "Chilled water outlet"
END_VISUALIZATION

// /Alarm_list
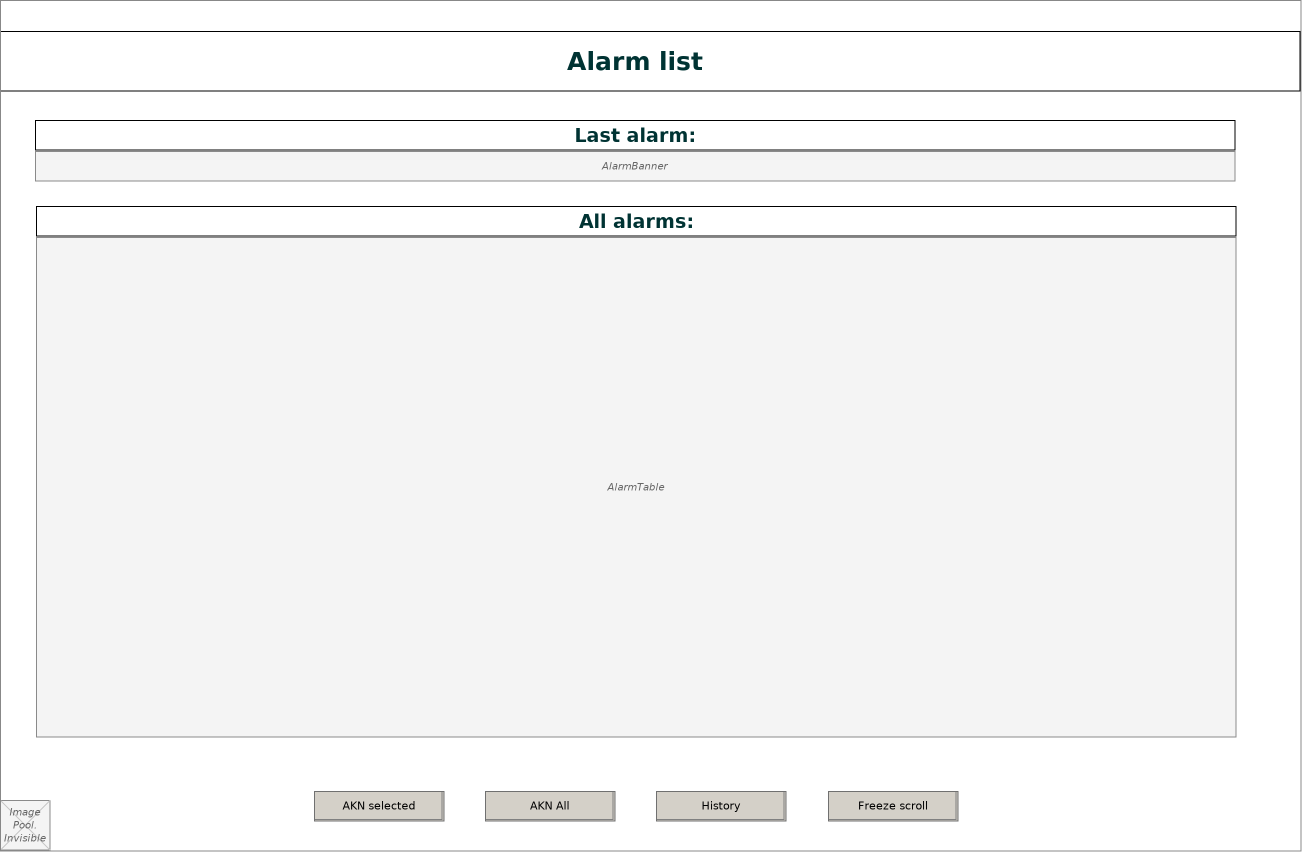
VISUALIZATION Alarm_list  // 1302x852
VAR
	AlarmACKButton : BOOL;
	AlarmACKAllButton : BOOL;
	AlarmHistoryButton : BOOL;
	AlarmFreezeButton : BOOL;
END_VAR
    AlarmTable (36,237 1200x500)
        p1521930926: __All
        p1663851261: __All
        p428520879: AlarmACKButton
        p2607059081: AlarmACKAllButton
        p3266827225: AlarmHistoryButton
        p3894972949: AlarmFreezeButton
    Button (314,791 130x30), "AKN selected"
        tap AlarmACKButton
    Button (485,791 130x30), "AKN All"
        tap AlarmACKAllButton
    Button (828,791 130x30), "Freeze scroll"
        toggle AlarmFreezeButton
    Button (656,791 130x30), "History"
        toggle AlarmHistoryButton
    Rectangle (0,31 1300x60)
    Label (247,33 776x56), "Alarm list"
    Rectangle (36,206 1200x30)
    Label (391,209 491x25), "All alarms:"
    Image (0,800 50x50), image: ImagePool.Invisible
    Rectangle (35,120 1200x30)
    Label (390,123 491x25), "Last alarm:"
    AlarmBanner (35,151 1200x30)
        p1521930926: __All
        p1663851261: __All
END_VISUALIZATION

// /Chiller1Menu
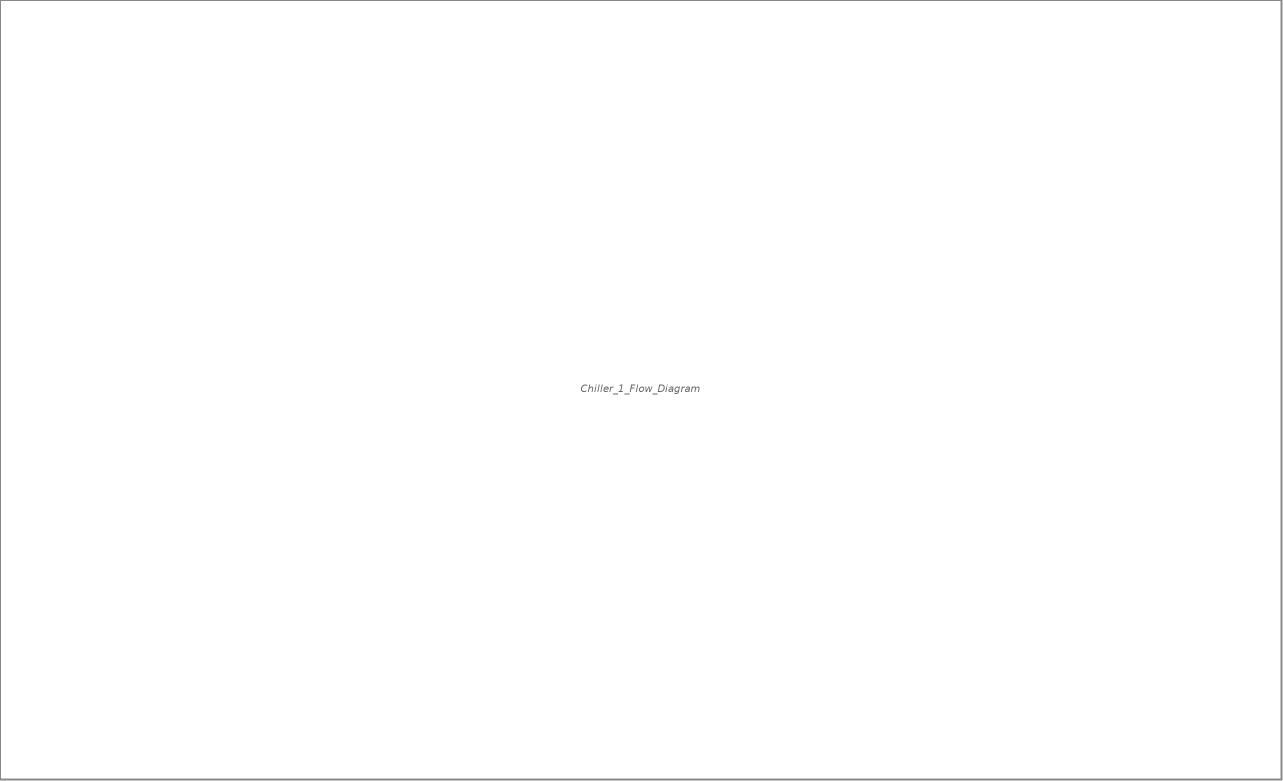
VISUALIZATION Chiller1Menu  // 1283x781
    TabControl (0,-2 1281x781)
        shows Chiller_1_Flow_Diagram()
        shows Chiller_1_Values()
        shows Chiller_1_Oil()
        shows Chiller_1_Alarm()
        shows Chiller_1_Trip()
        shows Chiller_1_VFD()
        [0]: TabTitle=Diagram
        [1]: TabTitle=Measured values
        [2]: TabTitle=Oil system
        [3]: TabTitle=Alarm
        [4]: TabTitle=Trip
END_VISUALIZATION

// /Chiller2Menu
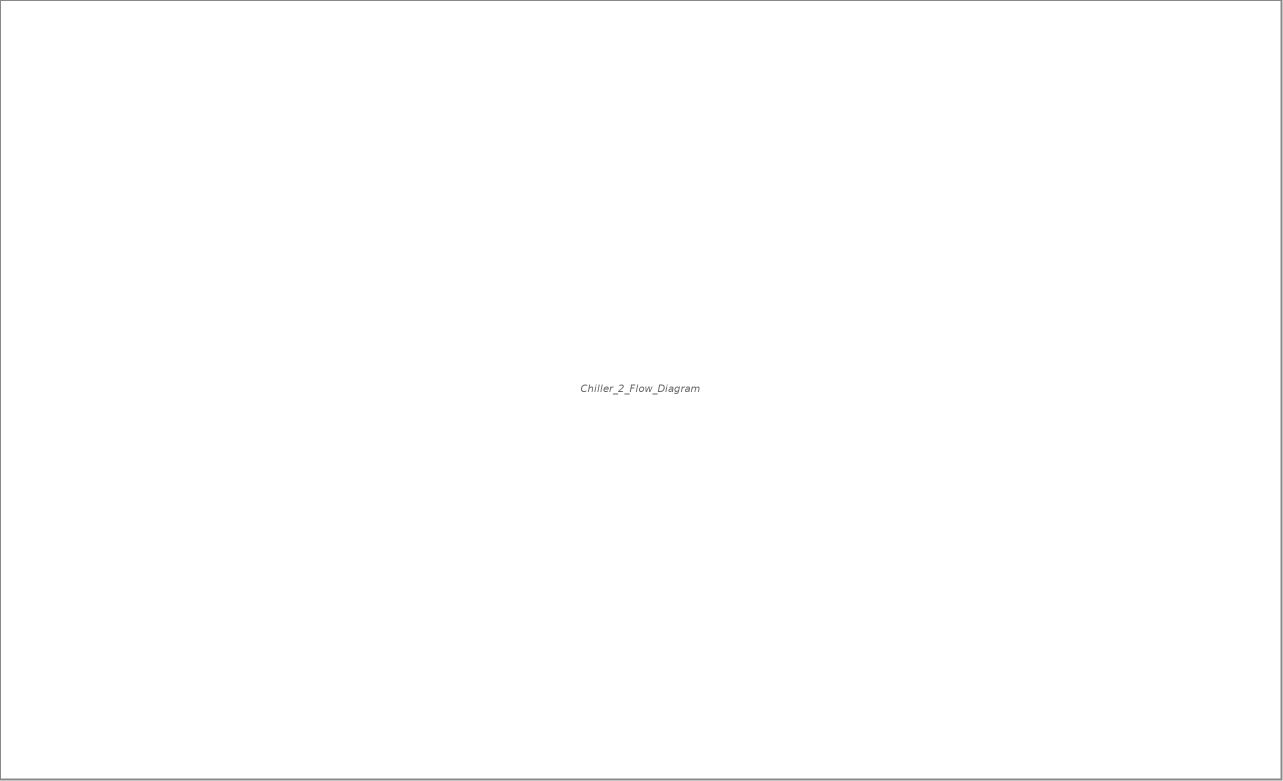
VISUALIZATION Chiller2Menu  // 1283x781
    TabControl (0,-2 1281x781)
        shows Chiller_2_Flow_Diagram()
        shows Chiller_2_Values()
        shows Chiller_2_Oil()
        shows Chiller_2_Alarm()
        shows Chiller_2_Trip()
        shows Chiller_1_Trip()
        [0]: TabTitle=Diagram
        [1]: TabTitle=Measured values
        [2]: TabTitle=Oil system
        [3]: TabTitle=Alarm
        [4]: TabTitle=Trip
        [5]: TabTitle=Trip
END_VISUALIZATION

// /Chiller3Menu
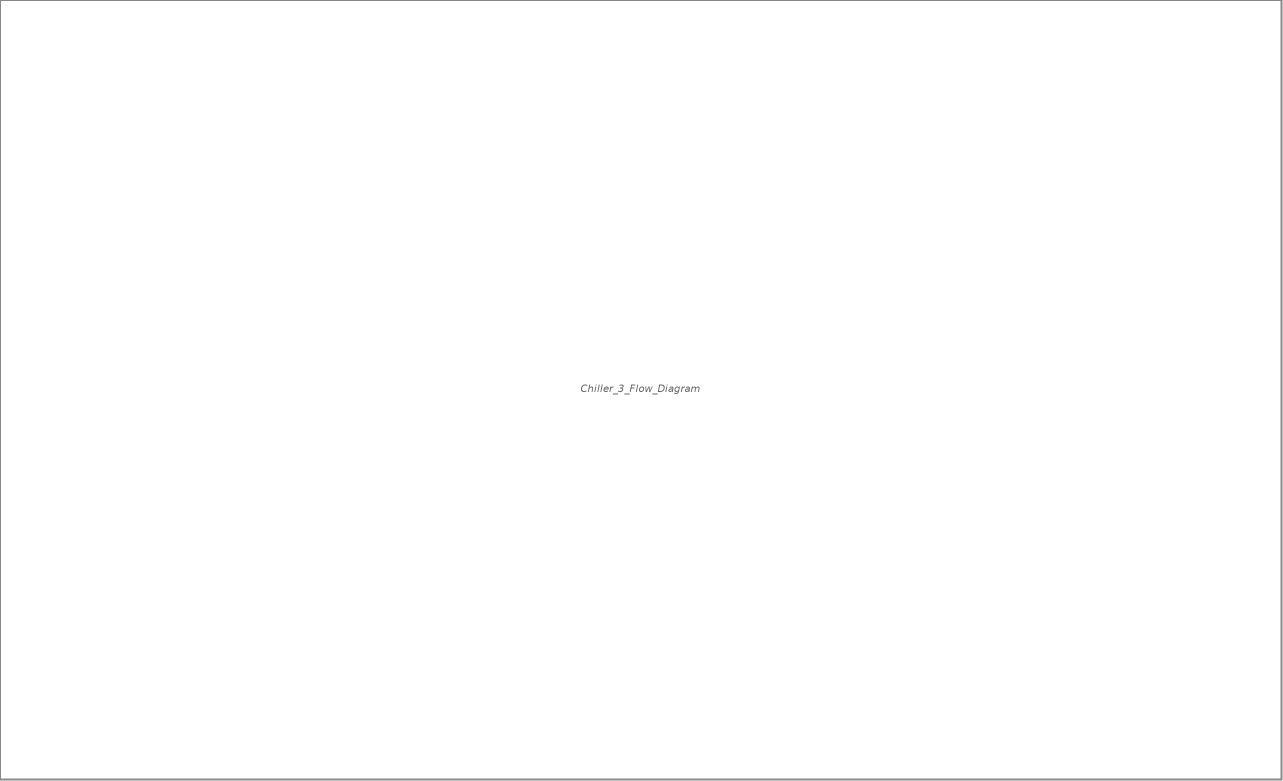
VISUALIZATION Chiller3Menu  // 1283x781
    TabControl (0,-2 1281x781)
        shows Chiller_3_Flow_Diagram()
        shows Chiller_3_Values()
        shows Chiller_3_Oil()
        shows Chiller_3_Alarm()
        shows Chiller_3_Trip()
        shows Chiller_1_Trip()
        [0]: TabTitle=Diagram
        [1]: TabTitle=Measured values
        [2]: TabTitle=Oil system
        [3]: TabTitle=Alarm
        [4]: TabTitle=Trip
        [5]: TabTitle=Trip
END_VISUALIZATION

// /Chiller4Menu
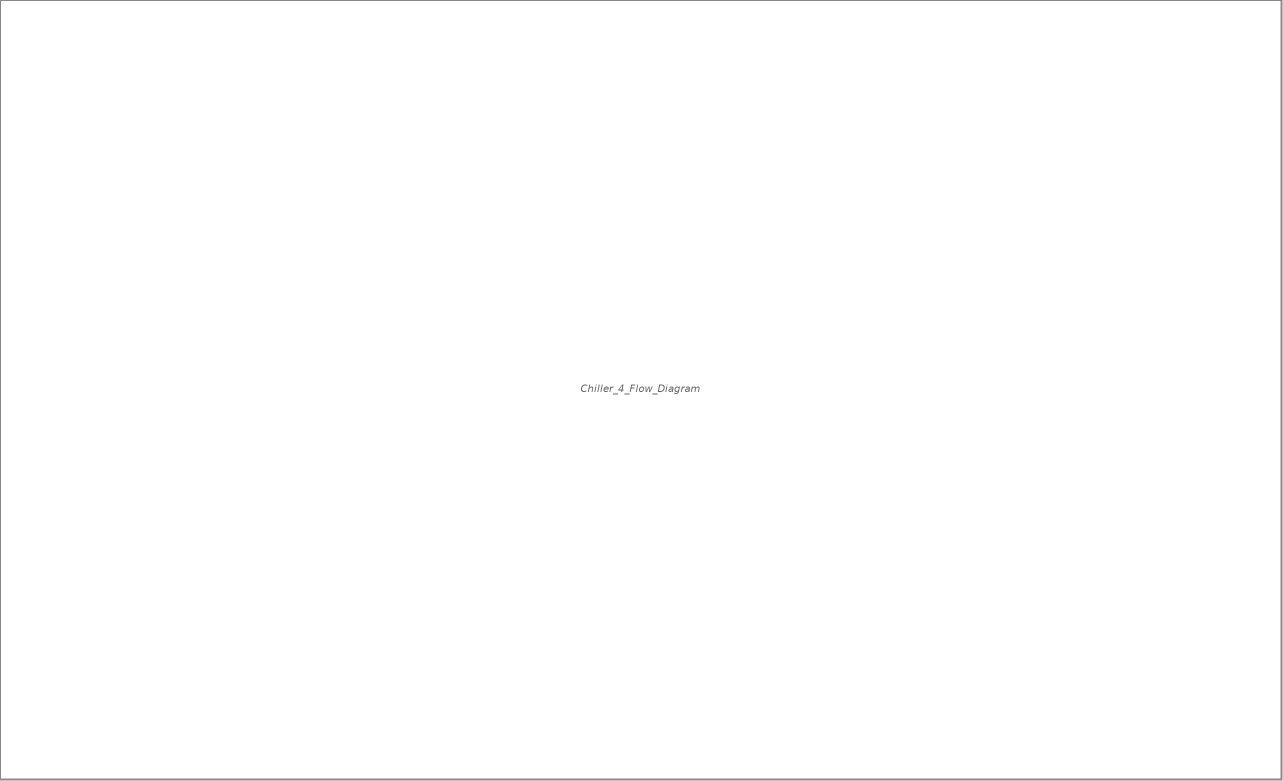
VISUALIZATION Chiller4Menu  // 1283x781
    TabControl (0,-2 1281x781)
        shows Chiller_4_Flow_Diagram()
        shows Chiller_4_Values()
        shows Chiller_4_Oil()
        shows Chiller_4_Alarm()
        shows Chiller_4_Trip()
        shows Chiller_1_Trip()
        [0]: TabTitle=Diagram
        [1]: TabTitle=Measured values
        [2]: TabTitle=Oil system
        [3]: TabTitle=Alarm
        [4]: TabTitle=Trip
        [5]: TabTitle=Trip
END_VISUALIZATION

// /Chiller_1_Alarm
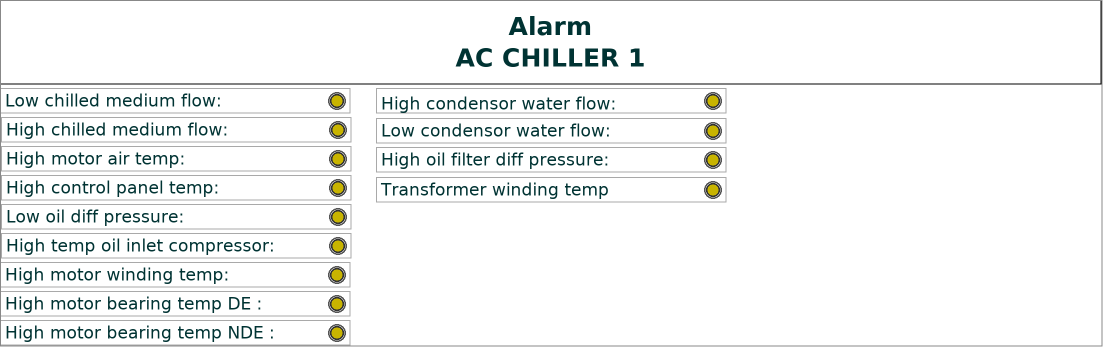
VISUALIZATION Chiller_1_Alarm  // 1103x347
    Rectangle (0,0 1101x84)
    Label (19,7 1063x70), "Alarm AC CHILLER 1"
    Rectangle (1,117 350x25)
    Label (3,119 314x21), "High chilled medium flow:"
    Lamp1 (327,120 22x20), variable: not.Chiller_1.A_High_chilled_medium_flow, style: Lamp-Lamp1-Yellow
    Rectangle (0,262 350x25)
    Label (2,264 314x21), "High motor winding temp:"
    Lamp1 (326,265 22x20), variable: not.Chiller_1.A_High_comp_motor_winding_temp, style: Lamp-Lamp1-Yellow
    Rectangle (0,291 350x25)
    Label (2,293 315x21), "High motor bearing temp DE :"
    Lamp1 (326,294 22x20), variable: not.Chiller_1.A_High_comp_mo_DE_bear_temp, style: Lamp-Lamp1-Yellow
    Rectangle (1,233 350x25)
    Label (3,235 312x21), "High temp oil inlet compressor:"
    Lamp1 (327,236 22x20), variable: not.Chiller_1.A_High_temp_oil_inlet_comp, style: Lamp-Lamp1-Yellow
    Rectangle (1,175 350x25)
    Label (3,177 309x21), "High control panel temp:"
    Lamp1 (327,178 22x20), variable: not.Chiller_1.A_High_control_panel_temp, style: Lamp-Lamp1-Yellow
    Rectangle (1,204 350x25)
    Label (3,206 315x21), "Low oil diff pressure:"
    Lamp1 (327,207 22x20), variable: not.Chiller_1.A_Low_oil_diff_pressure, style: Lamp-Lamp1-Yellow
    Rectangle (376,118 350x25)
    Label (378,120 320x21), "Low condensor water flow:"
    Lamp1 (702,121 22x20), variable: not.Chiller_1.A_Low_sea_water_flow, style: Lamp-Lamp1-Yellow
    Rectangle (376,147 350x25)
    Label (378,149 319x21), "High oil filter diff pressure:"
    Lamp1 (702,150 22x20), variable: not.Chiller_1.A_High_oil_filter_diff_press, style: Lamp-Lamp1-Yellow
    Rectangle (1,146 350x25)
    Label (3,148 314x21), "High motor air temp:"
    Lamp1 (327,149 22x20), variable: not.Chiller_1.A_High_motor_air_temp, style: Lamp-Lamp1-Yellow
    Rectangle (0,320 350x25)
    Label (2,322 315x21), "High motor bearing temp NDE :"
    Lamp1 (326,323 22x20), variable: not.Chiller_1.A_High_comp_mo_NDE_bear_temp, style: Lamp-Lamp1-Yellow
    Rectangle (0,88 350x25)
    Label (2,90 314x21), "Low chilled medium flow:"
    Lamp1 (326,91 22x20), variable: not.Chiller_1.A_Low_chilled_medium_flow, style: Lamp-Lamp1-Yellow
    Rectangle (376,88 350x25)
    Label (378,96 319x15), "High condensor water flow:"
    Lamp1 (702,91 22x20), variable: not.Chiller_1.A_High_condenser_flow, style: Lamp-Lamp1-Yellow
    Rectangle (376,177 350x25)
    Label (378,179 319x21), "Transformer winding temp"
    Lamp1 (702,180 22x20), variable: not.Chiller_1.A_Transformer_winding_temp, style: Lamp-Lamp1-Yellow
END_VISUALIZATION

// /Chiller_1_Alarm
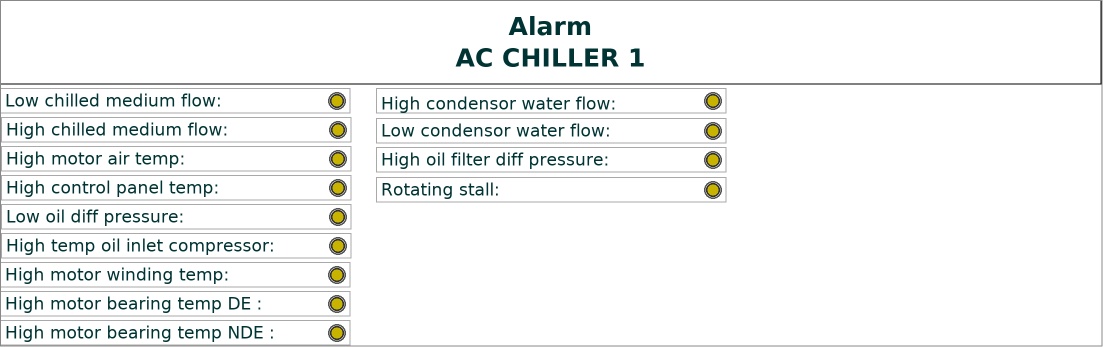
VISUALIZATION Chiller_1_Alarm  // 1103x347
    Rectangle (0,0 1101x84)
    Label (19,7 1063x70), "Alarm AC CHILLER 1"
    Rectangle (1,117 350x25)
    Label (3,119 314x21), "High chilled medium flow:"
    Lamp1 (327,120 22x20), variable: not.Chiller_1.A_High_chilled_medium_flow, style: Lamp-Lamp1-Yellow
    Rectangle (0,262 350x25)
    Label (2,264 314x21), "High motor winding temp:"
    Lamp1 (326,265 22x20), variable: not.Chiller_1.A_High_comp_motor_winding_temp, style: Lamp-Lamp1-Yellow
    Rectangle (0,291 350x25)
    Label (2,293 315x21), "High motor bearing temp DE :"
    Lamp1 (326,294 22x20), variable: not.Chiller_1.A_High_comp_mo_DE_bear_temp, style: Lamp-Lamp1-Yellow
    Rectangle (1,233 350x25)
    Label (3,235 312x21), "High temp oil inlet compressor:"
    Lamp1 (327,236 22x20), variable: not.Chiller_1.A_High_temp_oil_inlet_comp, style: Lamp-Lamp1-Yellow
    Rectangle (1,175 350x25)
    Label (3,177 309x21), "High control panel temp:"
    Lamp1 (327,178 22x20), variable: not.Chiller_1.A_High_control_panel_temp, style: Lamp-Lamp1-Yellow
    Rectangle (1,204 350x25)
    Label (3,206 315x21), "Low oil diff pressure:"
    Lamp1 (327,207 22x20), variable: not.Chiller_1.A_Low_oil_diff_pressure, style: Lamp-Lamp1-Yellow
    Rectangle (376,118 350x25)
    Label (378,120 320x21), "Low condensor water flow:"
    Lamp1 (702,121 22x20), variable: not.Chiller_1.A_Low_sea_water_flow, style: Lamp-Lamp1-Yellow
    Rectangle (376,147 350x25)
    Label (378,149 319x21), "High oil filter diff pressure:"
    Lamp1 (702,150 22x20), variable: not.Chiller_1.A_High_oil_filter_diff_press, style: Lamp-Lamp1-Yellow
    Rectangle (1,146 350x25)
    Label (3,148 314x21), "High motor air temp:"
    Lamp1 (327,149 22x20), variable: not.Chiller_1.A_High_motor_air_temp, style: Lamp-Lamp1-Yellow
    Rectangle (0,320 350x25)
    Label (2,322 315x21), "High motor bearing temp NDE :"
    Lamp1 (326,323 22x20), variable: not.Chiller_1.A_High_comp_mo_NDE_bear_temp, style: Lamp-Lamp1-Yellow
    Rectangle (0,88 350x25)
    Label (2,90 314x21), "Low chilled medium flow:"
    Lamp1 (326,91 22x20), variable: not.Chiller_1.A_Low_chilled_medium_flow, style: Lamp-Lamp1-Yellow
    Rectangle (376,88 350x25)
    Label (378,96 319x15), "High condensor water flow:"
    Lamp1 (702,91 22x20), variable: not.Chiller_1.A_High_condenser_flow, style: Lamp-Lamp1-Yellow
    Rectangle (376,177 350x25)
    Label (378,179 319x21), "Rotating stall:"
    Lamp1 (702,180 22x20), variable: not.Chiller_1.A_Rotating_stall, style: Lamp-Lamp1-Yellow
END_VISUALIZATION

